// SIMATIC STEP 7 (V5.x) project Daysil_Autoclav_v3

SYMBOL_TABLE
"AI-SENSOR-DATA"	DB 1	DB 1
"ORTAK_DATA"	DB 2	DB 2	// Ortak Veriler
"TIME_OTO_1_DB"	DB 5	SFB 4
"TIME_OTO_2_DB"	DB 6	SFB 4
"TIME_OTO_1_PROSES_DB"	DB 7	SFB 4
"TIME_OTO_2_PROSES_DB"	DB 8	SFB 4
"SURELER_DB"	DB 14	FB 3
"SAFETY_DB"	DB 15	FB 2
"KAZAN1_DATA"	DB 17	DB 17
"KAZAN2_DATA"	DB 18	DB 18	// KAZAN 2 BILGILERI
"JEN1_DATA"	DB 19	DB 19
"JEN2_DATA"	DB 20	DB 20
"JEN1_PID_DATA"	DB 21	DB 21
"JEN2_PID_DATA"	DB 22	DB 22
"KAZAN1_PID_DATA"	DB 23	DB 23	// KAZAN 1 PID BILGILERI
"KAZAN2_PID_DATA"	DB 24	DB 24	// KAZAN 2 PID BILGILERI
"JEN2_KONTROL_BLOGU_DB"	DB 51	FB 50
"JEN_1_PID_DB"	DB 69	FB 58
"JEN_2_PID_DB"	DB 70	FB 58
"OTOKLAV_1_DB"	DB 94	FB 94
"OTOKLAV_2_DB"	DB 95	FB 95
"FB98_DB"	DB 98	FB 98
"FB99_DB"	DB 99	FB 99
"HMI_DATA"	DB 100	DB 100	// Hmi arayuz verileri
"KAZAN_1_PID_DB"	DB 130	FB 58
"KAZAN_2_PID_DATA"	DB 231	FB 58
"MAINBLOCK"	FB 1	FB 1	// ANA PROGRAM BLOGU
"SAFETY"	FB 2	FB 2
"SURELER"	FB 3	FB 3
"TEST_BLOGU"	FB 5	FB 5
"KAZAN_ORTAK"	FB 20	FB 20
"KAZAN_PID_ORTAK"	FB 21	FB 21
"CONT_C"	FB 41	FB 41	// Continuous Control
"KAZAN_1_PID_KONTROL"	FB 47	FB 47
"KAZAN_2_PID_KONTROL"	FB 48	FB 48
"JEN1_PID_KONTROL"	FB 49	FB 49
"JEN2_PID_KONTROL"	FB 50	FB 50	// BUAHR JENERATÖR 2 PID
"TCONT_CP"	FB 58	FB 58	// temperature PID controller with pulse generator and self-tuning
"KAZAN_1_KONTROL"	FB 94	FB 94
"KAZAN_2_KONTROL"	FB 95	FB 95
"KAZAN1_KONTROL_BLOGU"	FB 96	FB 96
"KAZAN2_KONTROL_BLOGU"	FB 97	FB 97
"JEN1_KONTROL_BLOGU"	FB 98	FB 98
"JEN2_KONTROL_BLOGU"	FB 99	FB 99
"TIME_UNSCALE"	FC 1	FC 1
"O.Vana_AciklikHesaplama"	FC 2	FC 2	// Oransal vana aciklik orani hesaplama
"Int_To_S5Time"	FC 10	FC 10
"TIM_S5TI"	FC 40	FC 40	// IEC Time to S5 Time
"SCALE"	FC 105	FC 105	// Scaling Values
"UNSCALE"	FC 106	FC 106	// Unscaling Values
"KAZAN1_ACIL_STOP"	I 0.0	BOOL	// Acil Stop
"KAZAN1_START"	I 0.1	BOOL	// Kazan 1 Start
"KAZAN1_TRANSFER"	I 0.2	BOOL	// Kazan 1 Buhar Transferi
"KAZAN1_BOSALTIM"	I 0.3	BOOL	// Kazan 1 Bosaltim
"KAZAN1_KAPAK_SW"	I 0.4	BOOL	// Kazan 1 Kapak Kapandi
"KAZAN2_ACIL_STOP"	I 0.5	BOOL	// Kazan 2 Acil Stop
"KAZAN2_START"	I 0.6	BOOL	// Kazan 2 Start
"KAZAN2_TRANSFER"	I 0.7	BOOL	// Kazan 2 Buhar Transferi
"KAZAN2_BOSALTIM"	I 1.0	BOOL	// Kazan 2 Bosaltim
"KAZAN2_KAPAK_SW"	I 1.1	BOOL	// Kazan 2 Kapak Kapandi
"JEN1_STOP"	I 1.2	BOOL	// Jenerator 1 Stop
"JEN1_START"	I 1.3	BOOL	// Jenerator 1 Start
"JEN2_STOP"	I 1.4	BOOL	// Jenerator 2 Stop
"JEN2_START"	I 1.5	BOOL	// Jenerator 2 Start
"MANUEL"	I 1.6	BOOL	// Manuel Mod
"OTOMATIK"	I 1.7	BOOL	// Otomatik Mod
"JEN2_MOTOR_CALISTI"	I 2.0	BOOL
"JEN_1_MIN_SU_SEVIYESI"	I 3.0	BOOL
"JEN_2_MIN_SU_SEVIYESI"	I 3.1	BOOL
"0.1 SN."	M 0.0	BOOL
"0.2 SN."	M 0.1	BOOL
"0.4 SN."	M 0.2	BOOL
"0.5 SN."	M 0.3	BOOL
"0.8 SN."	M 0.4	BOOL
"1.0 SN."	M 0.5	BOOL
"1.6 SN."	M 0.6	BOOL
"2.0 SN."	M 0.7	BOOL
"Oto_1_Proses_BASLADI"	M 20.0	BOOL
"Oto_2_Proses_Basladi"	M 20.1	BOOL
"JEN2_CALIS_SURESI_BASLA"	M 22.0	BOOL
"JEN2_CALISTI_RIS"	M 22.1	BOOL
"JEN1_CALIS_SURESI_BASLA"	M 23.0	BOOL
"JEN1_CALISTI_RIS"	M 23.1	BOOL
"Jen1_Guvenlik_set_reset"	M 25.0	BOOL
"Jen2_Guvenlik_Set_Reset"	M 26.0	BOOL
"OTO_1_BEKLEME_BASLADI"	M 27.0	BOOL
"OTO_2_BEKLEME_BASLADI"	M 27.1	BOOL
"KAZAN_1_PID_MAN_ON"	M 35.0	BOOL
"KAZAN_2_MAN_ON"	M 37.0	BOOL
"TEST_START"	M 40.0	BOOL
"TEST_STOP"	M 40.1	BOOL
"TEST_OUT"	M 40.2	BOOL
"ALWAYS OFF"	M 100.0	BOOL	// ALWAYS OFF
"ALWAYS ON"	M 100.1	BOOL	// ALWAYS ON
"SET2_ULASMADI_SR"	M 101.0	BOOL
"SET2_ULASMADI_RIS"	M 101.1	BOOL
"JEN2_TCONT_MAN_ON"	M 155.0	BOOL
"Jen2_Stop_Trigger"	M 200.0	BOOL
"Jen2_Stop_Ris"	M 200.1	BOOL
"Jen2_Stop_Set_Mem"	M 200.2	BOOL
"JEN2_STOP_SET_RESET"	M 201.0	BOOL
"Sicaklik Dustu"	M 201.1	BOOL
"Ris_Jen2_Sicaklik_Dustu"	M 201.2	BOOL
"Rising_Sogutma"	M 201.3	BOOL
"Falling_Sogutma"	M 201.4	BOOL
"JEN1_STOP_SET_RESET"	M 202.0	BOOL
"START"	M 700.1	BOOL
"PID_START"	M 700.2	BOOL
"BRULOR_START"	M 700.3	BOOL
"SICAKLIK_1_OK"	M 700.5	BOOL
"SICAKLIK_2_OK"	M 700.6	BOOL
"BURLOR_MOTOR_START"	M 700.7	BOOL
"STOP"	M 701.1	BOOL
"100_DERECE_RIS"	M 750.0	BOOL
"Jen2_Ris"	M 750.4	BOOL
"Jen1_Ris"	M 750.5	BOOL
"BOS"	M 1000.0	BOOL
"O.VanaIlkAciklik"	MD 42	REAL	// Oransal vana ilk aciklik orani
"O.VanaKademeArtis"	MD 46	REAL	// Oransal vana kademeli artis orani
"PID BLOCK"	OB 35	OB 35	// PID BLOCK
"ZAMANHATASI"	OB 80	OB 80	// ZAMAN HATASI
"GERILIMHATASI"	OB 81	OB 81	// BESLEME GERILIMI HATASI
"HATAUYARISI"	OB 82	OB 82	// HATA UYARISI
"TAKMACIKARMAHATASI"	OB 83	OB 83	// TAKMA ÇIKARMA UYARISI
"CPUHARDWAREERROR"	OB 84	OB 84	// CPU HARDWARE ERROR
"PROGRAMHATASI"	OB 85	OB 85	// PROGRAM YURUTME HATASI
"RACKHATASI"	OB 86	OB 86	// RACK HATASI
"HABERLESMEHATASI"	OB 87	OB 87	// HABERLESME HATASI,
"COMPLETE RESTART"	OB 100	OB 100	// Complete Restart
"RESTART"	OB 101	OB 101	// Restart
"COLD RESTART"	OB 102	OB 102	// Cold Restart
"PROGRAMMINGERROR"	OB 121	OB 121	// PROGRAMLAMA HATASI
"MOD_ERR"	OB 122	OB 122	// Module Access Error
"KAZAN1_YESIL_LAMBA"	Q 0.0	BOOL	// Kazan 1 Yesil Lamba
"KAZAN1_KIRMIZI_LAMBA"	Q 0.1	BOOL	// Kazan 1 Kirmizi Lamba
"KAZAN1_DUDUK"	Q 0.2	BOOL	// Kazan 1 Duduk
"KAZAN1_BOSALTIM_VALFI"	Q 0.3	BOOL	// Kazan 1 Buhar Bosaltim
"KAZAN1_TRANS_BUT_LAMBASI"	Q 0.4	BOOL	// Kazan 1 Transfer Lambasi
"KAZAN1_EMN_VALFI_BOS"	Q 0.5	BOOL	// Kazan  1 Emniyet vantili bosaltim valfi
"KAZAN2_YESIL_LAMBA"	Q 0.6	BOOL	// Kazan 2 Yesil Lamba
"KAZAN2_KIRMIZI_LAMBA"	Q 0.7	BOOL	// Kazan 2 Kirmizi Lamba
"KAZAN2_DUDUK"	Q 1.0	BOOL	// Kazan 2 Duduk
"KAZAN2_BOSALTIM_VALFI"	Q 1.1	BOOL	// Kazan 2 Buhar Bosaltim
"KAZAN2_TRANS_BUT_LAMBASI"	Q 1.2	BOOL	// Kazan 2 Transfer Lambasi
"KAZAN2_EMN_VALFI_BOS"	Q 1.3	BOOL	// Kazan Emniyet vantili bosaltim valfi
"JEN_1_HAT_VANASI"	Q 1.4	BOOL
"JEN_1_PANO_STOP_LAMBASI"	Q 1.5	BOOL
"JEN_1_PANO_START_LAMBASI"	Q 1.6	BOOL
"JEN_2_HAT_VANASI"	Q 1.7	BOOL
"JEN_2_PANO_STOP_LAMBASI"	Q 2.0	BOOL
"JEN_2_PANO_START_LAMBASI"	Q 2.1	BOOL
"PANO_OTO_MAN_BUTON_LAMBA"	Q 2.2	BOOL
"PANO_ALARM"	Q 2.3	BOOL
"JEN_1_BRULOR"	Q 2.4	BOOL
"JEN_1_POMPA"	Q 2.5	BOOL
"JEN_2_BRULOR_OUT"	Q 2.6	BOOL
"JEN_2_SU_POM_OUT"	Q 2.7	BOOL
"TON"	SFB 4	SFB 4	// Generate an On Delay
"TIME_TCK"	SFC 64	SFC 64	// Read the System Time
"delay_300ms_1"	T 8	TIMER
"500ms_delay1"	T 10	TIMER
"1s Delay"	T 11	TIMER
"Pisim_Suresi"	T 12	TIMER
"500ms_delay"	T 13	TIMER
"s_offt_7s_delay"	T 14	TIMER
"tm_adim1_pid_basla_delay"	T 16	TIMER
"500ms_delay_kazan_2"	T 20	TIMER
"1ms_delay_kazan_2"	T 21	TIMER
"kazan_2_pisirme_delay"	T 22	TIMER
"kazan_2_500ms_delay"	T 23	TIMER
"kazan_2_7s_delay"	T 24	TIMER
"Delay_500ms_Jen2"	T 30	TIMER
"DELAY_1S_JEN_HATA"	T 33	TIMER
"DELAY_300MS"	T 42	TIMER
"DELAY_500MS_1"	T 43	TIMER
"DELAY_5S_pompa"	T 44	TIMER
"OTO_2_DELAY_BITIS"	T 50	TIMER
"OTO_1_DELAY_PISIM_BITTI"	T 51	TIMER
"DELAY_ADIM5_BEKLE"	T 52	TIMER
"DELAY_ADIM5_BEKLE2"	T 53	TIMER
"TIM_SET2_ULASMADI"	T 57	TIMER
"VAT_1"	VAT 1	
END_SYMBOL_TABLE

FUNCTION_BLOCK "MAINBLOCK"	// FB 1
VERSION : 0.1
BEGIN
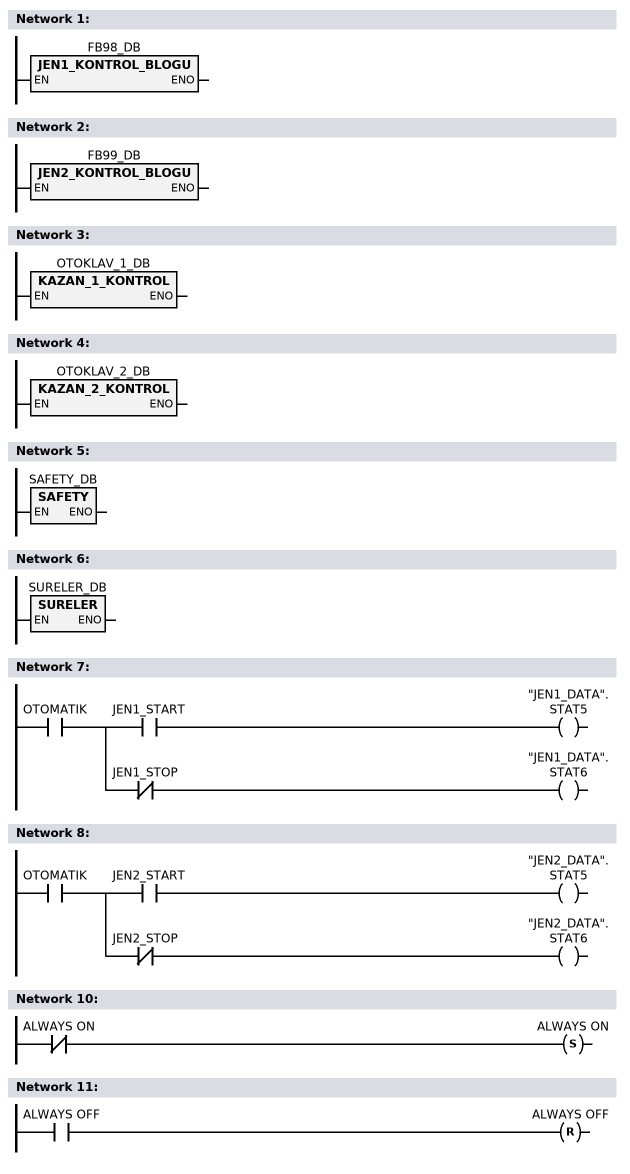
NETWORK
TITLE =
      CALL  "JEN1_KONTROL_BLOGU" , "FB98_DB";
      NOP   0;
NETWORK
TITLE =
      CALL  "JEN2_KONTROL_BLOGU" , "FB99_DB";
      NOP   0;
NETWORK
TITLE =
      CALL  "KAZAN_1_KONTROL" , "OTOKLAV_1_DB";
      NOP   0;
NETWORK
TITLE =
      CALL  "KAZAN_2_KONTROL" , "OTOKLAV_2_DB";
      NOP   0;
NETWORK
TITLE =
      CALL  "SAFETY" , "SAFETY_DB";
      NOP   0;
NETWORK
TITLE =
      CALL  "SURELER" , "SURELER_DB";
      NOP   0;
NETWORK
TITLE =
      A     "OTOMATIK";
      =     L 0.0;
      A     L 0.0;
      A     "JEN1_START";
      =     "JEN1_DATA".STAT5;
      A     L 0.0;
      AN    "JEN1_STOP";
      =     "JEN1_DATA".STAT6;
NETWORK
TITLE =
      A     "OTOMATIK";
      =     L 0.0;
      A     L 0.0;
      A     "JEN2_START";
      =     "JEN2_DATA".STAT5;
      A     L 0.0;
      AN    "JEN2_STOP";
      =     "JEN2_DATA".STAT6;
NETWORK
TITLE =
NETWORK
TITLE =
      AN    "ALWAYS ON";
      S     "ALWAYS ON";
NETWORK
TITLE =
      A     "ALWAYS OFF";
      R     "ALWAYS OFF";
NETWORK
TITLE =
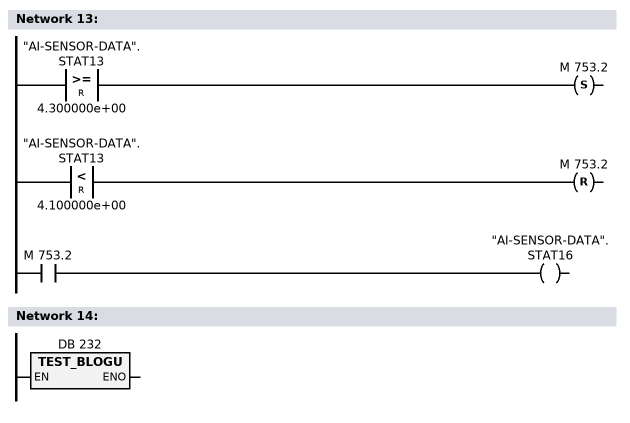
NETWORK
TITLE =
      A(;
      L     "AI-SENSOR-DATA".STAT13;
      L     4.300000e+00;
      >=R;
      );
      S     M 753.2;
      A(;
      L     "AI-SENSOR-DATA".STAT13;
      L     4.100000e+00;
      <R;
      );
      R     M 753.2;
      A     M 753.2;
      =     "AI-SENSOR-DATA".STAT16;
NETWORK
TITLE =
      CALL  "TEST_BLOGU" , DB 232;
      NOP   0;
END_FUNCTION_BLOCK

FUNCTION_BLOCK "SAFETY"	// FB 2
VERSION : 0.1
BEGIN
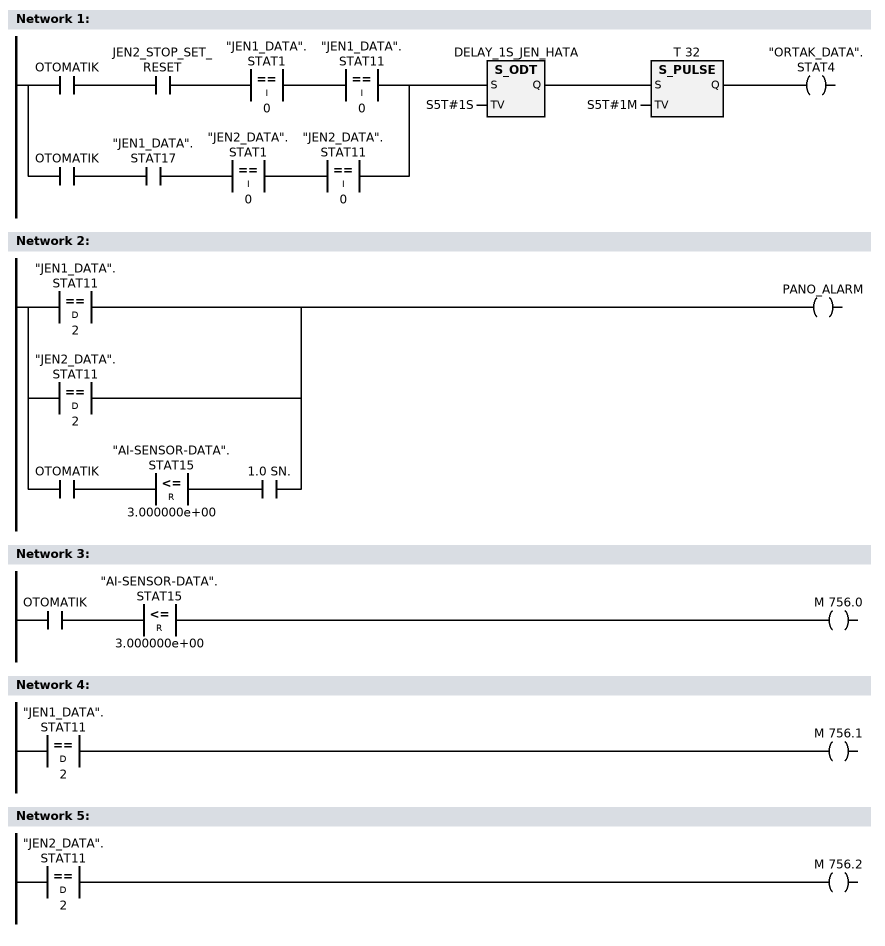
NETWORK
TITLE =
      A(;
      A(;
      A     "OTOMATIK";
      A     "JEN2_STOP_SET_RESET";
      A(;
      L     "JEN1_DATA".STAT1;
      L     0;
      ==I;
      );
      A(;
      L     "JEN1_DATA".STAT11;
      L     0;
      ==I;
      );
      O;
      A     "OTOMATIK";
      A     "JEN1_DATA".STAT17;
      A(;
      L     "JEN2_DATA".STAT1;
      L     0;
      ==I;
      );
      A(;
      L     "JEN2_DATA".STAT11;
      L     0;
      ==I;
      );
      );
      L     S5T#1S;
      SD    "DELAY_1S_JEN_HATA";
      NOP   0;
      NOP   0;
      NOP   0;
      A     "DELAY_1S_JEN_HATA";
      );
      L     S5T#1M;
      SP    T 32;
      NOP   0;
      NOP   0;
      NOP   0;
      A     T 32;
      =     "ORTAK_DATA".STAT4;
NETWORK
TITLE =
      O(;
      L     "JEN1_DATA".STAT11;
      L     2;
      ==D;
      );
      O(;
      L     "JEN2_DATA".STAT11;
      L     2;
      ==D;
      );
      O;
      A     "OTOMATIK";
      A(;
      L     "AI-SENSOR-DATA".STAT15;
      L     3.000000e+00;
      <=R;
      );
      A     "1.0 SN.";
      =     "PANO_ALARM";
NETWORK
TITLE =
      A     "OTOMATIK";
      A(;
      L     "AI-SENSOR-DATA".STAT15;
      L     3.000000e+00;
      <=R;
      );
      =     M 756.0;
NETWORK
TITLE =
      L     "JEN1_DATA".STAT11;
      L     2;
      ==D;
      =     M 756.1;
NETWORK
TITLE =
      L     "JEN2_DATA".STAT11;
      L     2;
      ==D;
      =     M 756.2;
END_FUNCTION_BLOCK

FUNCTION_BLOCK "SURELER"	// FB 3
VERSION : 0.1
BEGIN
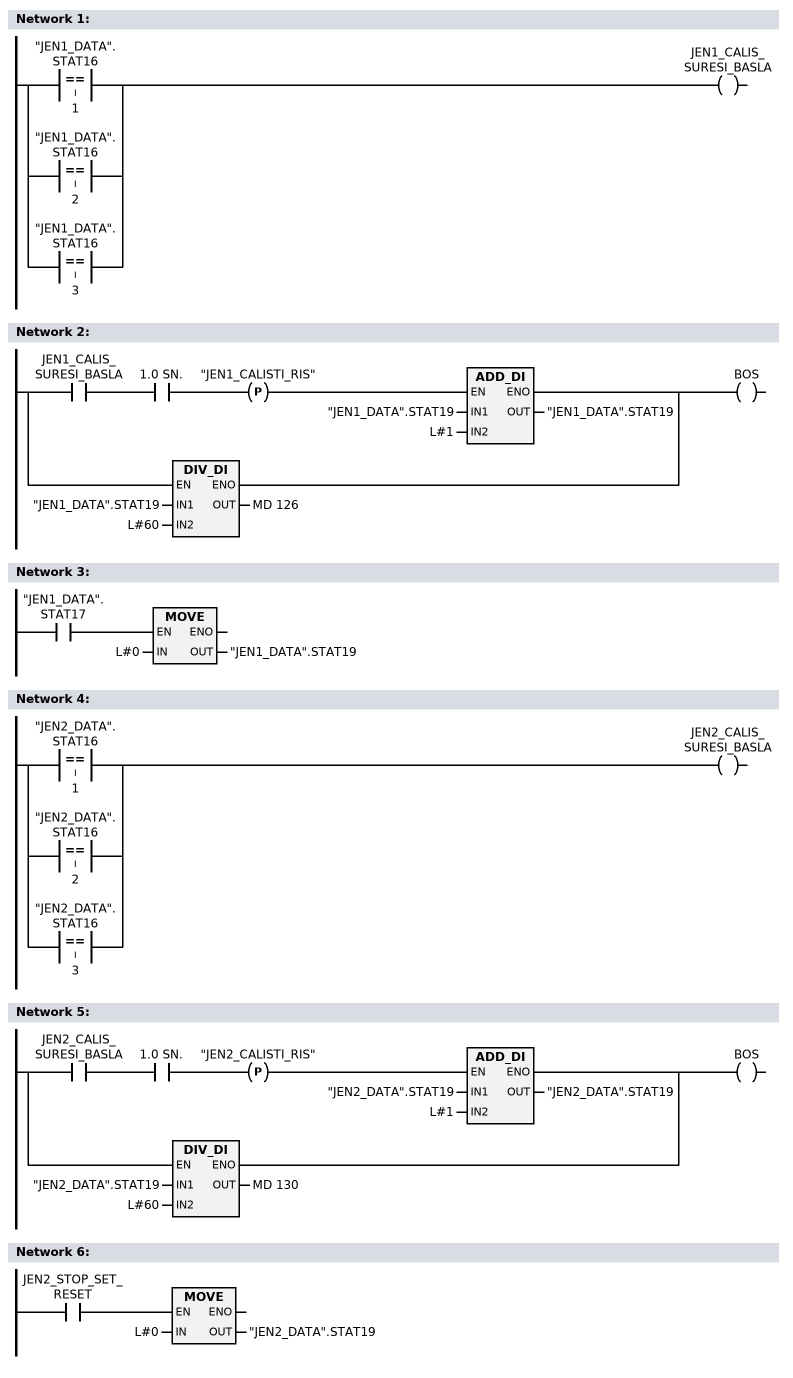
NETWORK
TITLE =
      O(;
      L     "JEN1_DATA".STAT16;
      L     1;
      ==I;
      );
      O(;
      L     "JEN1_DATA".STAT16;
      L     2;
      ==I;
      );
      O(;
      L     "JEN1_DATA".STAT16;
      L     3;
      ==I;
      );
      =     "JEN1_CALIS_SURESI_BASLA";
NETWORK
TITLE =
      O(;
      A     "JEN1_CALIS_SURESI_BASLA";
      A     "1.0 SN.";
      FP    "JEN1_CALISTI_RIS";
      JNB   _001;
      L     "JEN1_DATA".STAT19;
      L     L#1;
      +D;
      T     "JEN1_DATA".STAT19;
      AN    OV;
      SAVE;
      CLR;
_001: A     BR;
      );
      O(;
      L     "JEN1_DATA".STAT19;
      L     L#60;
      /D;
      T     MD 126;
      AN    OV;
      SAVE;
      CLR;
      A     BR;
      );
      =     "BOS";
NETWORK
TITLE =
      A     "JEN1_DATA".STAT17;
      JNB   _002;
      L     L#0;
      T     "JEN1_DATA".STAT19;
_002: NOP   0;
NETWORK
TITLE =
      O(;
      L     "JEN2_DATA".STAT16;
      L     1;
      ==I;
      );
      O(;
      L     "JEN2_DATA".STAT16;
      L     2;
      ==I;
      );
      O(;
      L     "JEN2_DATA".STAT16;
      L     3;
      ==I;
      );
      =     "JEN2_CALIS_SURESI_BASLA";
NETWORK
TITLE =
      O(;
      A     "JEN2_CALIS_SURESI_BASLA";
      A     "1.0 SN.";
      FP    "JEN2_CALISTI_RIS";
      JNB   _003;
      L     "JEN2_DATA".STAT19;
      L     L#1;
      +D;
      T     "JEN2_DATA".STAT19;
      AN    OV;
      SAVE;
      CLR;
_003: A     BR;
      );
      O(;
      L     "JEN2_DATA".STAT19;
      L     L#60;
      /D;
      T     MD 130;
      AN    OV;
      SAVE;
      CLR;
      A     BR;
      );
      =     "BOS";
NETWORK
TITLE =
      A     "JEN2_STOP_SET_RESET";
      JNB   _004;
      L     L#0;
      T     "JEN2_DATA".STAT19;
_004: NOP   0;
NETWORK
TITLE =
      O(;
      A(;
      A     "KAZAN1_DATA".STAT19;
      =     L 0.0;
      BLD   103;
      BLD   9;
      =     L 5.0;
      CDB;
      OPN   DI 5;
      TAR2  LD 1;
      A     L 0.0;
      =     DIX 0.0;
      L     L#82800000;
      T     DID 2;
      LAR2  P#DBX 0.0;
      UC    "TON";
      LAR2  LD 1;
      L     DID 8;
      OPN   DI 17;
      T     DID 42;
      OPN   DI 5;
      CDB;
      BLD   10;
      A     BR;
      );
      JNB   _005;
      CALL  "TIME_UNSCALE" (
           $1                       := "KAZAN1_DATA".STAT20,
           $2                       := "KAZAN1_DATA".STAT3,
           $3                       := "KAZAN1_DATA".STAT21);
_005: A     BR;
      );
      O(;
      L     "KAZAN1_DATA".STAT21;
      L     60;
      /D;
      T     MD 118;
      AN    OV;
      SAVE;
      CLR;
      A     BR;
      );
      =     "BOS";
NETWORK
TITLE =
      O(;
      A(;
      A     "KAZAN2_DATA".STAT19;
      =     L 0.0;
      BLD   103;
      BLD   9;
      =     L 5.0;
      CDB;
      OPN   DI 6;
      TAR2  LD 1;
      A     L 0.0;
      =     DIX 0.0;
      L     L#82800000;
      T     DID 2;
      LAR2  P#DBX 0.0;
      UC    "TON";
      LAR2  LD 1;
      L     DID 8;
      OPN   DI 18;
      T     DID 42;
      OPN   DI 6;
      CDB;
      BLD   10;
      A     BR;
      );
      JNB   _006;
      CALL  "TIME_UNSCALE" (
           $1                       := "KAZAN2_DATA".STAT20,
           $2                       := "KAZAN2_DATA".STAT3,
           $3                       := "KAZAN2_DATA".STAT21);
_006: A     BR;
      );
      O(;
      L     "KAZAN2_DATA".STAT21;
      L     60;
      /D;
      T     MD 122;
      AN    OV;
      SAVE;
      CLR;
      A     BR;
      );
      =     "BOS";
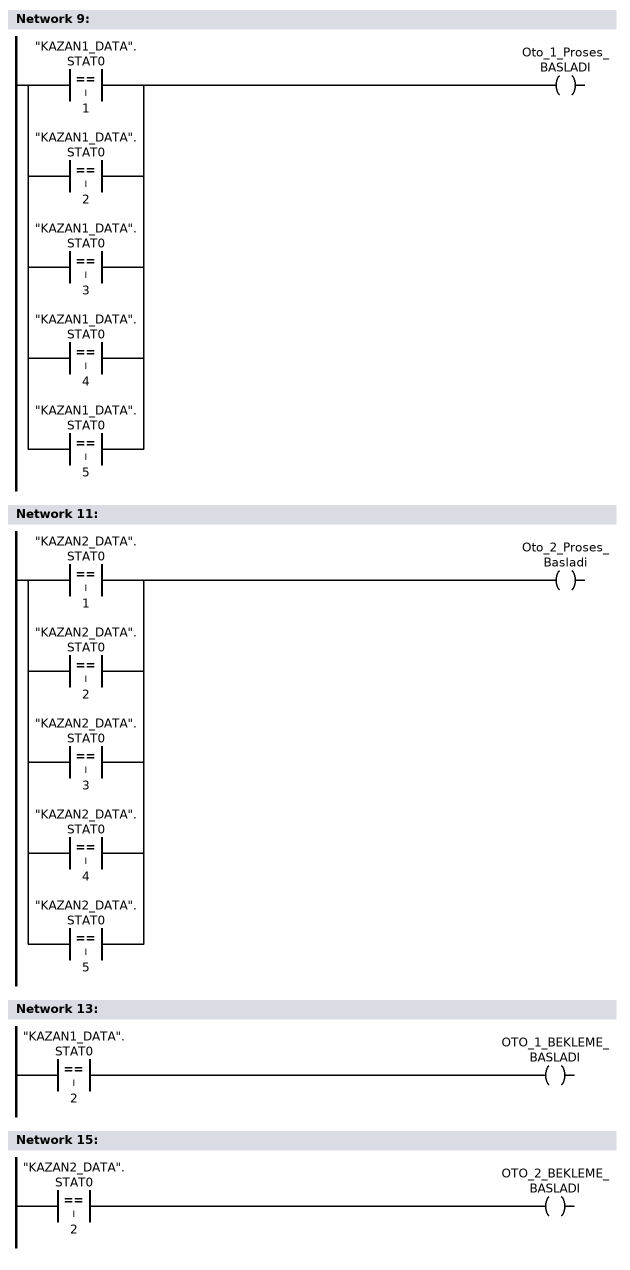
NETWORK
TITLE =
      O(;
      L     "KAZAN1_DATA".STAT0;
      L     1;
      ==I;
      );
      O(;
      L     "KAZAN1_DATA".STAT0;
      L     2;
      ==I;
      );
      O(;
      L     "KAZAN1_DATA".STAT0;
      L     3;
      ==I;
      );
      O(;
      L     "KAZAN1_DATA".STAT0;
      L     4;
      ==I;
      );
      O(;
      L     "KAZAN1_DATA".STAT0;
      L     5;
      ==I;
      );
      =     "Oto_1_Proses_BASLADI";
NETWORK
TITLE =
      O(;
      A(;
      A     "Oto_1_Proses_BASLADI";
      =     L 0.0;
      BLD   103;
      BLD   9;
      =     L 5.0;
      CDB;
      OPN   DI 7;
      TAR2  LD 1;
      A     L 0.0;
      =     DIX 0.0;
      L     L#82800000;
      T     DID 2;
      LAR2  P#DBX 0.0;
      UC    "TON";
      LAR2  LD 1;
      L     DID 8;
      OPN   DI 17;
      T     DID 50;
      OPN   DI 7;
      CDB;
      BLD   10;
      A     BR;
      );
      JNB   _007;
      L     "KAZAN1_DATA".STAT22;
      L     1000;
      /D;
      T     "KAZAN1_DATA".STAT23;
      AN    OV;
      SAVE;
      CLR;
_007: A     BR;
      );
      O(;
      L     "KAZAN1_DATA".STAT23;
      L     60;
      /D;
      T     MD 110;
      AN    OV;
      SAVE;
      CLR;
      A     BR;
      );
      =     "BOS";
NETWORK
TITLE =
      O(;
      L     "KAZAN2_DATA".STAT0;
      L     1;
      ==I;
      );
      O(;
      L     "KAZAN2_DATA".STAT0;
      L     2;
      ==I;
      );
      O(;
      L     "KAZAN2_DATA".STAT0;
      L     3;
      ==I;
      );
      O(;
      L     "KAZAN2_DATA".STAT0;
      L     4;
      ==I;
      );
      O(;
      L     "KAZAN2_DATA".STAT0;
      L     5;
      ==I;
      );
      =     "Oto_2_Proses_Basladi";
NETWORK
TITLE =
      O(;
      A(;
      A     "Oto_2_Proses_Basladi";
      =     L 0.0;
      BLD   103;
      BLD   9;
      =     L 5.0;
      CDB;
      OPN   DI 8;
      TAR2  LD 1;
      A     L 0.0;
      =     DIX 0.0;
      L     L#82800000;
      T     DID 2;
      LAR2  P#DBX 0.0;
      UC    "TON";
      LAR2  LD 1;
      L     DID 8;
      OPN   DI 18;
      T     DID 50;
      OPN   DI 8;
      CDB;
      BLD   10;
      A     BR;
      );
      JNB   _008;
      L     "KAZAN2_DATA".STAT22;
      L     1000;
      /D;
      T     "KAZAN2_DATA".STAT23;
      AN    OV;
      SAVE;
      CLR;
_008: A     BR;
      );
      O(;
      L     "KAZAN2_DATA".STAT23;
      L     60;
      /D;
      T     MD 114;
      AN    OV;
      SAVE;
      CLR;
      A     BR;
      );
      =     "BOS";
NETWORK
TITLE =
      L     "KAZAN1_DATA".STAT0;
      L     2;
      ==I;
      =     "OTO_1_BEKLEME_BASLADI";
NETWORK
TITLE =
      A(;
      A     "OTO_1_BEKLEME_BASLADI";
      =     L 0.0;
      BLD   103;
      BLD   9;
      =     L 5.0;
      CDB;
      OPN   DI 9;
      TAR2  LD 1;
      A     L 0.0;
      =     DIX 0.0;
      L     L#82800000;
      T     DID 2;
      LAR2  P#DBX 0.0;
      UC    "TON";
      LAR2  LD 1;
      L     DID 8;
      OPN   DI 17;
      T     DID 58;
      OPN   DI 9;
      CDB;
      BLD   10;
      A     BR;
      );
      JNB   _009;
      L     "KAZAN1_DATA".STAT24;
      L     1000;
      /D;
      T     "KAZAN1_DATA".STAT25;
_009: NOP   0;
NETWORK
TITLE =
      L     "KAZAN2_DATA".STAT0;
      L     2;
      ==I;
      =     "OTO_2_BEKLEME_BASLADI";
NETWORK
TITLE =
      A(;
      A     "OTO_2_BEKLEME_BASLADI";
      =     L 0.0;
      BLD   103;
      BLD   9;
      =     L 5.0;
      CDB;
      OPN   DI 10;
      TAR2  LD 1;
      A     L 0.0;
      =     DIX 0.0;
      L     L#82800000;
      T     DID 2;
      LAR2  P#DBX 0.0;
      UC    "TON";
      LAR2  LD 1;
      L     DID 8;
      OPN   DI 18;
      T     DID 58;
      OPN   DI 10;
      CDB;
      BLD   10;
      A     BR;
      );
      JNB   _00a;
      L     "KAZAN2_DATA".STAT24;
      L     1000;
      /D;
      T     "KAZAN2_DATA".STAT25;
_00a: NOP   0;
END_FUNCTION_BLOCK

FUNCTION_BLOCK "TEST_BLOGU"	// FB 5
VERSION : 0.1
BEGIN
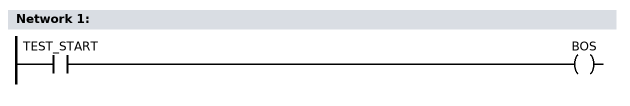
NETWORK
TITLE =
      A     "TEST_START";
      =     "BOS";
END_FUNCTION_BLOCK

FUNCTION_BLOCK "KAZAN_ORTAK"	// FB 20
VERSION : 0.1
VAR_INPUT
  IN0 : BOOL ;
  IN1 : BOOL ;
  IN2 : BOOL ;
  IN3 : BOOL ;
  IN4 : BOOL ;
  IN5 : BOOL ;
  IN6 : BOOL ;
  IN7 : BOOL ;
  IN8 : BOOL ;
  IN9 : S5TIME ;
  IN10 : INT ;
  IN11 : REAL ;
  IN12 : REAL ;
  IN13 : TIMER ;
  IN14 : TIMER ;
  IN15 : TIMER ;
  IN16 : TIMER ;
  IN17 : TIMER ;
  IN18 : REAL ;
  IN19 : REAL ;
  IN20 : REAL ;
  IN21 : REAL ;
  IN22 : INT ;
  IN23 : BOOL ;
  IN24 : BOOL ;
  IN25 : BLOCK_DB ;
  IN26 : BOOL ;
  IN27 : BOOL ;
  IN28 : REAL ;
  IN29 : TIMER ;
  IN30 : TIMER ;
  IN31 : TIMER ;
  IN32 : TIMER ;
END_VAR
VAR_OUTPUT
  OUT33 : BOOL ;
  OUT34 : BOOL ;
  OUT35 : BOOL ;
  OUT36 : BOOL ;
  OUT37 : BOOL ;
  OUT38 : REAL ;
  OUT39 : BOOL ;
  OUT40 : WORD ;
  OUT41 : REAL ;
  OUT42 : BOOL ;
  OUT43 : BOOL ;
  OUT44 : WORD ;
  OUT45 : REAL ;
  OUT46 : BOOL ;
  OUT47 : BOOL ;
  OUT48 : BOOL ;
  OUT49 : BOOL ;
END_VAR
VAR_IN_OUT
  IO50 : INT ;
END_VAR
VAR
  STAT51 : INT ;
  STAT52 : BOOL ;
  STAT53 : BOOL ;
  STAT54 : REAL ;
  STAT55 : BOOL ;
  STAT56 : REAL  := 1.000000e+001;
  STAT57 : REAL ;
  STAT58 : BOOL ;
  STAT59 : REAL ;
  STAT60 : REAL ;
  STAT61 : BOOL ;
  STAT62 : BOOL ;
  STAT63 : BOOL ;
  STAT64 : BOOL ;
  STAT65 : WORD ;
  STAT66 : REAL ;
  STAT67 : WORD ;
  STAT68 : REAL ;
  STAT69 : BOOL ;
  STAT70 : BOOL ;
  STAT71 : BOOL ;
  STAT72 : REAL ;
  STAT73 : TIME ;
  STAT74 : BOOL ;
  STAT75 : BOOL ;
  STAT76 : BOOL ;
  STAT77 : BOOL ;
  STAT78 : BOOL ;
END_VAR
VAR_TEMP
  tKademe : STRUCT
   Bir : REAL ;
   Iki : REAL ;
   Uc : REAL ;
   Dort : REAL ;
   Bes : REAL ;
   Alti : REAL ;
   Yedi : REAL ;
  END_STRUCT ;
END_VAR
BEGIN
NETWORK
TITLE =
      A(;
      A(;
      A     "ALWAYS OFF";
      =     L 28.0;
      BLD   103;
      CALL  "SCALE" (
           $1                       := #IN10,
           $2                       := #IN18,
           $3                       := #IN19,
           $4                       := L 28.0,
           $5                       := #STAT65,
           $6                       := #STAT66);
      A     BR;
      );
      JNB   _001;
      L     #STAT65;
      T     #OUT40;
      SET;
      SAVE;
      CLR;
_001: A     BR;
      );
      JNB   _002;
      L     #STAT66;
      T     #OUT41;
_002: NOP   0;
NETWORK
TITLE =
      A(;
      A(;
      A     "ALWAYS OFF";
      =     L 28.0;
      BLD   103;
      CALL  "SCALE" (
           $1                       := #IN22,
           $2                       := #IN20,
           $3                       := #IN21,
           $4                       := L 28.0,
           $5                       := #STAT67,
           $6                       := #STAT68);
      A     BR;
      );
      JNB   _003;
      L     #STAT67;
      T     #OUT44;
      SET;
      SAVE;
      CLR;
_003: A     BR;
      );
      JNB   _004;
      L     #STAT68;
      T     #OUT45;
_004: NOP   0;
NETWORK
TITLE =
      A(;
      A     "OTOMATIK";
      A     #IN0;
      A     "AI-SENSOR-DATA".STAT16;
      L     S5T#200MS;
      T     LD 28;
      TAK;
      T     LD 32;
      L     #IN13;
      T     LW 36;
      L     LD 32;
      L     LD 28;
      SD    T [LW 36];
      NOP   0;
      NOP   0;
      NOP   0;
      T     LD 28;
      TAK;
      T     LD 32;
      L     #IN13;
      T     LW 36;
      L     LD 32;
      L     LD 28;
      A     T [LW 36];
      );
      A     #IN4;
      A     #IN1;
      A(;
      L     #IO50;
      L     0;
      ==I;
      );
      JNB   _005;
      L     1;
      T     #IO50;
      SET;
      SAVE;
      CLR;
_005: A     BR;
      S     #STAT69;
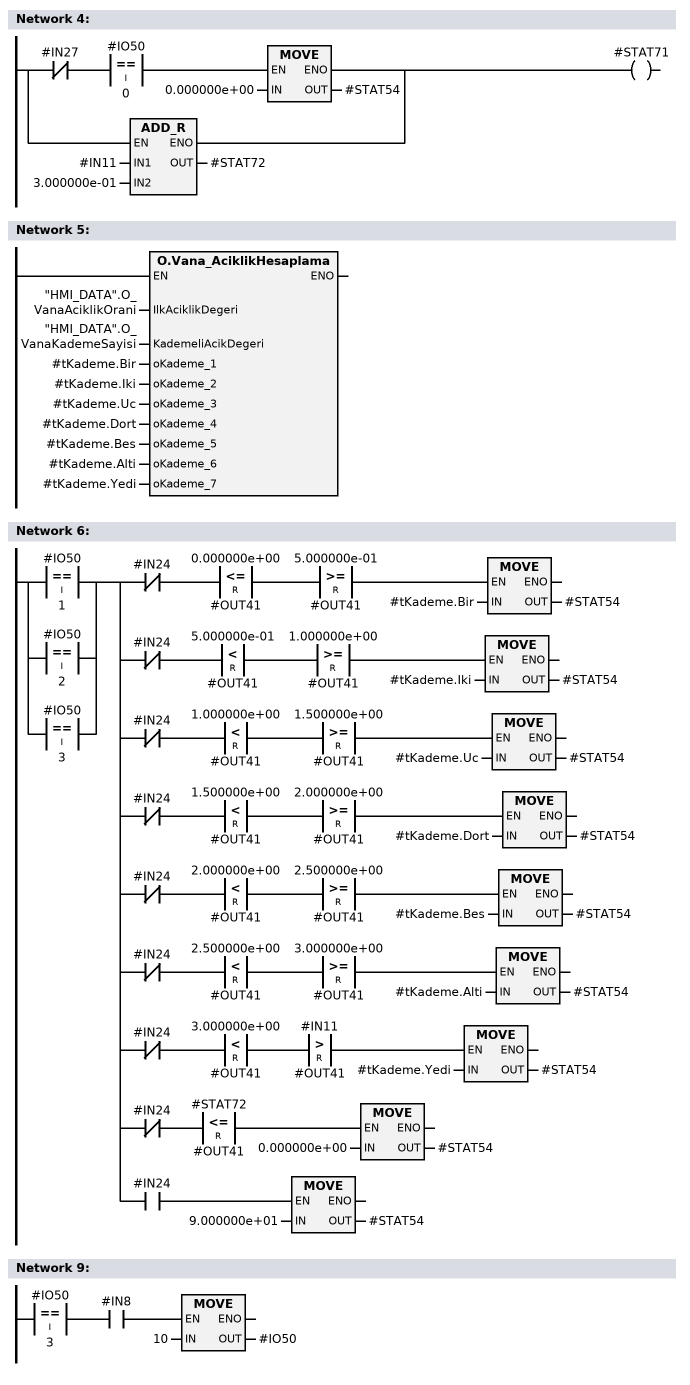
NETWORK
TITLE =
      O(;
      AN    #IN27;
      A(;
      L     #IO50;
      L     0;
      ==I;
      );
      JNB   _006;
      L     0.000000e+00;
      T     #STAT54;
      SET;
      SAVE;
      CLR;
_006: A     BR;
      );
      O(;
      L     #IN11;
      L     3.000000e-01;
      +R;
      T     #STAT72;
      AN    OV;
      SAVE;
      CLR;
      A     BR;
      );
      =     #STAT71;
NETWORK
TITLE =
      CALL  "O.Vana_AciklikHesaplama" (
           IlkAciklikDegeri         := "HMI_DATA".O_VanaAciklikOrani,
           KademeliAcikDegeri       := "HMI_DATA".O_VanaKademeSayisi,
           oKademe_1                := #tKademe.Bir,
           oKademe_2                := #tKademe.Iki,
           oKademe_3                := #tKademe.Uc,
           oKademe_4                := #tKademe.Dort,
           oKademe_5                := #tKademe.Bes,
           oKademe_6                := #tKademe.Alti,
           oKademe_7                := #tKademe.Yedi);
      NOP   0;
NETWORK
TITLE =
      O(;
      L     #IO50;
      L     1;
      ==I;
      );
      O(;
      L     #IO50;
      L     2;
      ==I;
      );
      O(;
      L     #IO50;
      L     3;
      ==I;
      );
      =     L 28.0;
      A     L 28.0;
      AN    #IN24;
      A(;
      L     0.000000e+00;
      L     #OUT41;
      <=R;
      );
      A(;
      L     5.000000e-01;
      L     #OUT41;
      >=R;
      );
      JNB   _007;
      L     #tKademe.Bir;
      T     #STAT54;
_007: NOP   0;
      A     L 28.0;
      AN    #IN24;
      A(;
      L     5.000000e-01;
      L     #OUT41;
      <R;
      );
      A(;
      L     1.000000e+00;
      L     #OUT41;
      >=R;
      );
      JNB   _008;
      L     #tKademe.Iki;
      T     #STAT54;
_008: NOP   0;
      A     L 28.0;
      AN    #IN24;
      A(;
      L     1.000000e+00;
      L     #OUT41;
      <R;
      );
      A(;
      L     1.500000e+00;
      L     #OUT41;
      >=R;
      );
      JNB   _009;
      L     #tKademe.Uc;
      T     #STAT54;
_009: NOP   0;
      A     L 28.0;
      AN    #IN24;
      A(;
      L     1.500000e+00;
      L     #OUT41;
      <R;
      );
      A(;
      L     2.000000e+00;
      L     #OUT41;
      >=R;
      );
      JNB   _00a;
      L     #tKademe.Dort;
      T     #STAT54;
_00a: NOP   0;
      A     L 28.0;
      AN    #IN24;
      A(;
      L     2.000000e+00;
      L     #OUT41;
      <R;
      );
      A(;
      L     2.500000e+00;
      L     #OUT41;
      >=R;
      );
      JNB   _00b;
      L     #tKademe.Bes;
      T     #STAT54;
_00b: NOP   0;
      A     L 28.0;
      AN    #IN24;
      A(;
      L     2.500000e+00;
      L     #OUT41;
      <R;
      );
      A(;
      L     3.000000e+00;
      L     #OUT41;
      >=R;
      );
      JNB   _00c;
      L     #tKademe.Alti;
      T     #STAT54;
_00c: NOP   0;
      A     L 28.0;
      AN    #IN24;
      A(;
      L     3.000000e+00;
      L     #OUT41;
      <R;
      );
      A(;
      L     #IN11;
      L     #OUT41;
      >R;
      );
      JNB   _00d;
      L     #tKademe.Yedi;
      T     #STAT54;
_00d: NOP   0;
      A     L 28.0;
      AN    #IN24;
      A(;
      L     #STAT72;
      L     #OUT41;
      <=R;
      );
      JNB   _00e;
      L     0.000000e+00;
      T     #STAT54;
_00e: NOP   0;
      A     L 28.0;
      A     #IN24;
      JNB   _00f;
      L     9.000000e+01;
      T     #STAT54;
_00f: NOP   0;
NETWORK
TITLE =
      L     #IO50;
      L     1;
      ==I;
      =     L 28.0;
      A(;
      A     L 28.0;
      A     #STAT58;
      L     #IN9;
      T     LD 29;
      TAK;
      T     LD 33;
      L     #IN15;
      T     LW 37;
      L     LD 33;
      L     LD 29;
      SD    T [LW 37];
      NOP   0;
      NOP   0;
      NOP   0;
      T     LD 29;
      TAK;
      T     LD 33;
      L     #IN15;
      T     LW 37;
      L     LD 33;
      L     LD 29;
      A     T [LW 37];
      );
      JNB   _010;
      L     2;
      T     #IO50;
_010: NOP   0;
      A     L 28.0;
      A(;
      O(;
      L     #OUT41;
      L     #IN11;
      >=R;
      );
      O     #STAT58;
      );
      =     #STAT58;
NETWORK
TITLE =
      L     #IO50;
      L     2;
      ==I;
      =     L 28.0;
      A     L 28.0;
      L     S5T#5M;
      T     LD 29;
      TAK;
      T     LD 33;
      L     #IN31;
      T     LW 37;
      L     LD 33;
      L     LD 29;
      SD    T [LW 37];
      NOP   0;
      NOP   0;
      NOP   0;
      NOP   0;
      A     L 28.0;
      A     #IN2;
      JNB   _011;
      L     3;
      T     #IO50;
_011: NOP   0;
      A     L 28.0;
      A     #IN3;
      JNB   _012;
      L     4;
      T     #IO50;
_012: NOP   0;
NETWORK
TITLE =
      A(;
      L     #IO50;
      L     3;
      ==I;
      );
      A     #IN8;
      JNB   _013;
      L     10;
      T     #IO50;
_013: NOP   0;
NETWORK
TITLE =
      L     #IO50;
      L     10;
      ==I;
      =     L 28.0;
      A     L 28.0;
      JNB   _014;
      L     9.000000e+01;
      T     #STAT54;
      SET;
      SAVE;
      CLR;
_014: A     BR;
      =     #OUT39;
      A(;
      A     L 28.0;
      L     S5T#23S;
      T     LD 29;
      TAK;
      T     LD 33;
      L     #IN16;
      T     LW 37;
      L     LD 33;
      L     LD 29;
      SD    T [LW 37];
      NOP   0;
      NOP   0;
      NOP   0;
      T     LD 29;
      TAK;
      T     LD 33;
      L     #IN16;
      T     LW 37;
      L     LD 33;
      L     LD 29;
      A     T [LW 37];
      );
      JNB   _015;
      L     4;
      T     #IO50;
_015: NOP   0;
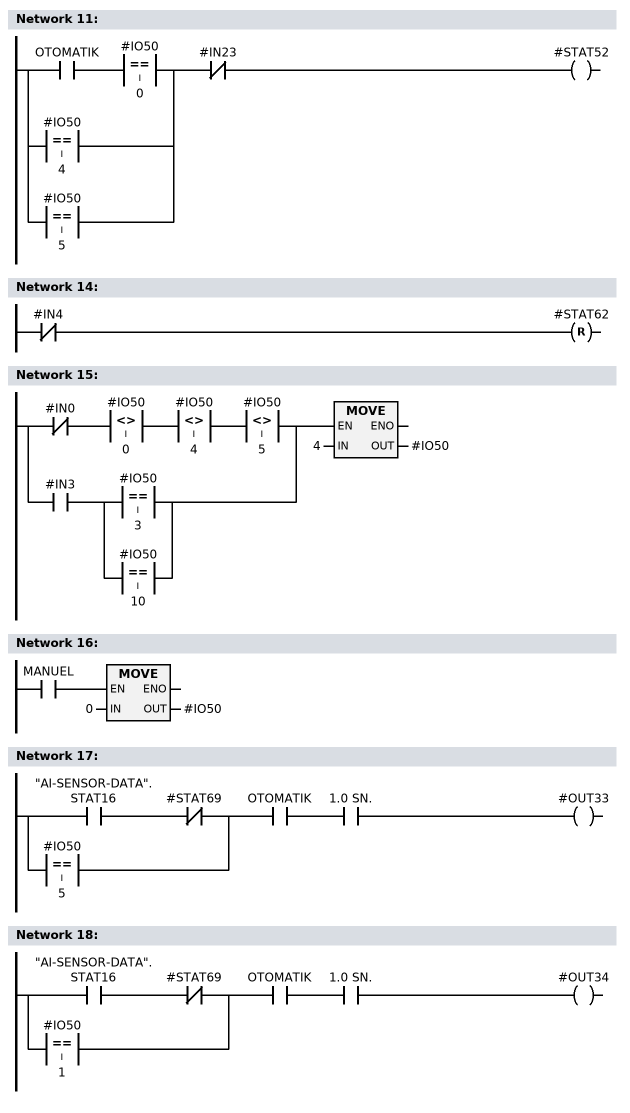
NETWORK
TITLE =
      A(;
      A     "OTOMATIK";
      A(;
      L     #IO50;
      L     0;
      ==I;
      );
      O(;
      L     #IO50;
      L     4;
      ==I;
      );
      O(;
      L     #IO50;
      L     5;
      ==I;
      );
      );
      AN    #IN23;
      =     #STAT52;
NETWORK
TITLE =
      L     #IO50;
      L     4;
      ==I;
      =     L 28.0;
      A     L 28.0;
      JNB   _016;
      L     0.000000e+00;
      T     #STAT54;
_016: NOP   0;
      A     L 28.0;
      BLD   102;
      =     #STAT70;
      A     L 28.0;
      A(;
      L     #OUT41;
      L     1.000000e-01;
      <=R;
      );
      =     L 28.1;
      A     L 28.1;
      BLD   102;
      S     #STAT62;
      A(;
      A     L 28.1;
      L     S5T#5S;
      T     LD 29;
      TAK;
      T     LD 33;
      L     #IN29;
      T     LW 37;
      L     LD 33;
      L     LD 29;
      SD    T [LW 37];
      NOP   0;
      NOP   0;
      NOP   0;
      T     LD 29;
      TAK;
      T     LD 33;
      L     #IN29;
      T     LW 37;
      L     LD 33;
      L     LD 29;
      A     T [LW 37];
      );
      JNB   _017;
      L     5;
      T     #IO50;
_017: NOP   0;
NETWORK
TITLE =
      A(;
      A(;
      L     #IO50;
      L     5;
      ==I;
      );
      L     S5T#1S;
      T     LD 28;
      TAK;
      T     LD 32;
      L     #IN30;
      T     LW 36;
      L     LD 32;
      L     LD 28;
      SD    T [LW 36];
      NOP   0;
      NOP   0;
      NOP   0;
      T     LD 28;
      TAK;
      T     LD 32;
      L     #IN30;
      T     LW 36;
      L     LD 32;
      L     LD 28;
      A     T [LW 36];
      );
      AN    #IN4;
      JNB   _018;
      L     0;
      T     #IO50;
_018: NOP   0;
NETWORK
TITLE =
      AN    #IN4;
      R     #STAT62;
NETWORK
TITLE =
      A(;
      AN    #IN0;
      A(;
      L     #IO50;
      L     0;
      <>I;
      );
      A(;
      L     #IO50;
      L     4;
      <>I;
      );
      A(;
      L     #IO50;
      L     5;
      <>I;
      );
      O;
      A     #IN3;
      A(;
      O(;
      L     #IO50;
      L     3;
      ==I;
      );
      O(;
      L     #IO50;
      L     10;
      ==I;
      );
      );
      );
      JNB   _019;
      L     4;
      T     #IO50;
_019: NOP   0;
NETWORK
TITLE =
      A     "MANUEL";
      JNB   _01a;
      L     0;
      T     #IO50;
_01a: NOP   0;
NETWORK
TITLE =
      A(;
      A     "AI-SENSOR-DATA".STAT16;
      AN    #STAT69;
      O(;
      L     #IO50;
      L     5;
      ==I;
      );
      );
      A     "OTOMATIK";
      A     "1.0 SN.";
      =     #OUT33;
NETWORK
TITLE =
      A(;
      A     "AI-SENSOR-DATA".STAT16;
      AN    #STAT69;
      O(;
      L     #IO50;
      L     1;
      ==I;
      );
      );
      A     "OTOMATIK";
      A     "1.0 SN.";
      =     #OUT34;
NETWORK
TITLE =
      A(;
      A(;
      L     #IO50;
      L     2;
      ==I;
      );
      A     "1.0 SN.";
      O(;
      A(;
      O(;
      L     #IO50;
      L     3;
      ==I;
      );
      O(;
      L     #IO50;
      L     10;
      ==I;
      );
      );
      AN    #OUT39;
      L     S5T#5M;
      T     LD 28;
      TAK;
      T     LD 32;
      L     #IN32;
      T     LW 36;
      L     LD 32;
      L     LD 28;
      SD    T [LW 36];
      NOP   0;
      NOP   0;
      NOP   0;
      T     LD 28;
      TAK;
      T     LD 32;
      L     #IN32;
      T     LW 36;
      L     LD 32;
      L     LD 28;
      A     T [LW 36];
      );
      );
      A     "OTOMATIK";
      =     #OUT35;
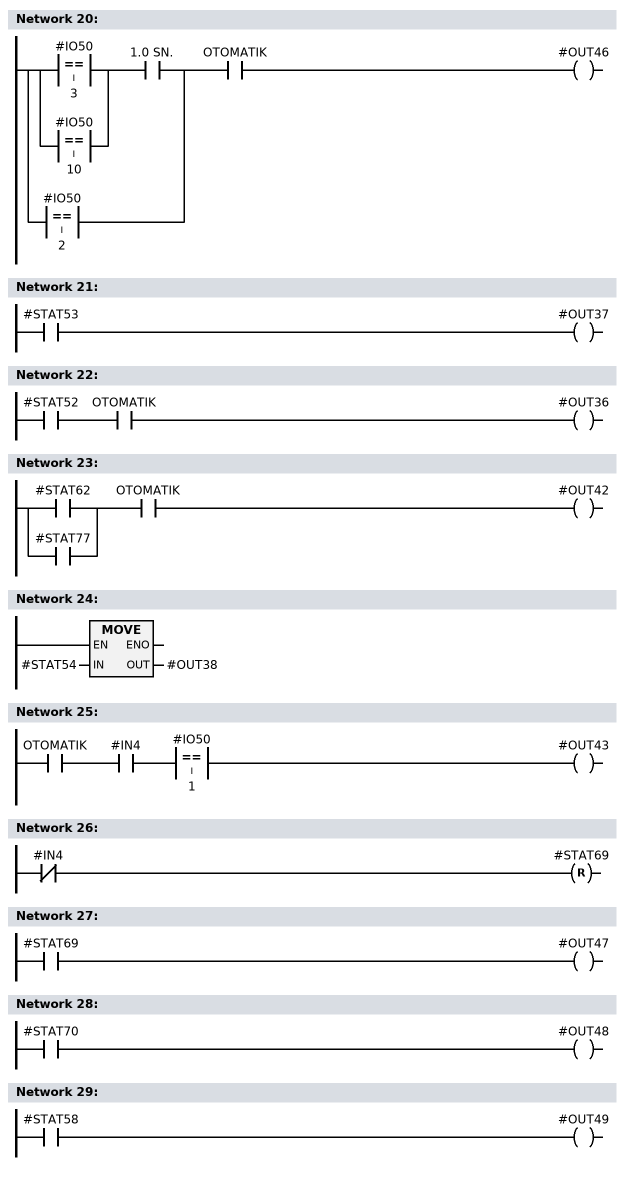
NETWORK
TITLE =
      A(;
      A(;
      O(;
      L     #IO50;
      L     3;
      ==I;
      );
      O(;
      L     #IO50;
      L     10;
      ==I;
      );
      );
      A     "1.0 SN.";
      O(;
      L     #IO50;
      L     2;
      ==I;
      );
      );
      A     "OTOMATIK";
      =     #OUT46;
NETWORK
TITLE =
      A     #STAT53;
      =     #OUT37;
NETWORK
TITLE =
      A     #STAT52;
      A     "OTOMATIK";
      =     #OUT36;
NETWORK
TITLE =
      A(;
      O     #STAT62;
      O     #STAT77;
      );
      A     "OTOMATIK";
      =     #OUT42;
NETWORK
TITLE =
      L     #STAT54;
      T     #OUT38;
      NOP   0;
NETWORK
TITLE =
      A     "OTOMATIK";
      A     #IN4;
      A(;
      L     #IO50;
      L     1;
      ==I;
      );
      =     #OUT43;
NETWORK
TITLE =
      AN    #IN4;
      R     #STAT69;
NETWORK
TITLE =
      A     #STAT69;
      =     #OUT47;
NETWORK
TITLE =
      A     #STAT70;
      =     #OUT48;
NETWORK
TITLE =
      A     #STAT58;
      =     #OUT49;
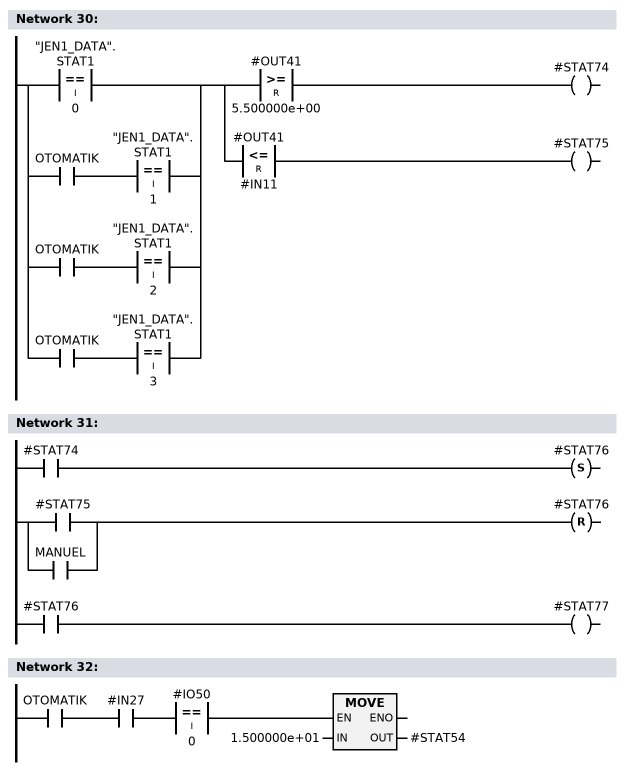
NETWORK
TITLE =
      O(;
      L     "JEN1_DATA".STAT1;
      L     0;
      ==I;
      );
      O;
      A     "OTOMATIK";
      A(;
      L     "JEN1_DATA".STAT1;
      L     1;
      ==I;
      );
      O;
      A     "OTOMATIK";
      A(;
      L     "JEN1_DATA".STAT1;
      L     2;
      ==I;
      );
      O;
      A     "OTOMATIK";
      A(;
      L     "JEN1_DATA".STAT1;
      L     3;
      ==I;
      );
      =     L 28.0;
      A     L 28.0;
      A(;
      L     #OUT41;
      L     5.500000e+00;
      >=R;
      );
      =     #STAT74;
      A     L 28.0;
      A(;
      L     #OUT41;
      L     #IN11;
      <=R;
      );
      =     #STAT75;
NETWORK
TITLE =
      A     #STAT74;
      S     #STAT76;
      A(;
      O     #STAT75;
      O     "MANUEL";
      );
      R     #STAT76;
      A     #STAT76;
      =     #STAT77;
NETWORK
TITLE =
      A     "OTOMATIK";
      A     #IN27;
      A(;
      L     #IO50;
      L     0;
      ==I;
      );
      JNB   _01b;
      L     1.500000e+01;
      T     #STAT54;
_01b: NOP   0;
END_FUNCTION_BLOCK

// FB 41: know-how protected block, not included

FUNCTION_BLOCK "KAZAN_1_PID_KONTROL"	// FB 47
VERSION : 0.1
BEGIN
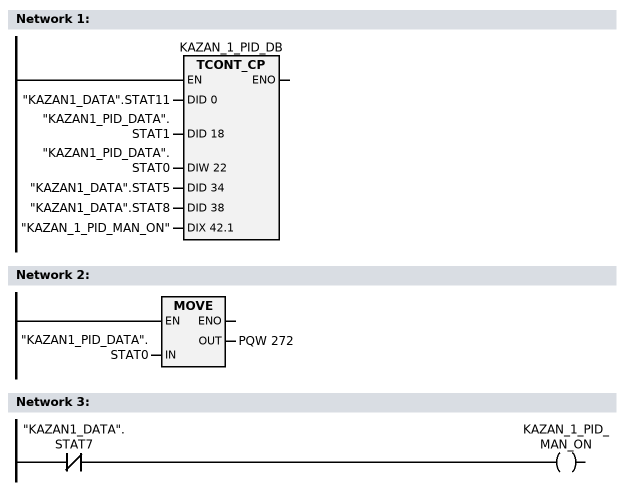
NETWORK
TITLE =
      CALL  "TCONT_CP" , "KAZAN_1_PID_DB" (
           DID 0                    := "KAZAN1_DATA".STAT11,
           DID 18                   := "KAZAN1_PID_DATA".STAT1,
           DIW 22                   := "KAZAN1_PID_DATA".STAT0,
           DID 34                   := "KAZAN1_DATA".STAT5,
           DID 38                   := "KAZAN1_DATA".STAT8,
           DIX 42.1                 := "KAZAN_1_PID_MAN_ON");
      NOP   0;
NETWORK
TITLE =
      L     "KAZAN1_PID_DATA".STAT0;
      T     PQW 272;
      NOP   0;
NETWORK
TITLE =
      AN    "KAZAN1_DATA".STAT7;
      =     "KAZAN_1_PID_MAN_ON";
NETWORK
TITLE =
END_FUNCTION_BLOCK

FUNCTION_BLOCK "KAZAN_2_PID_KONTROL"	// FB 48
VERSION : 0.1
BEGIN
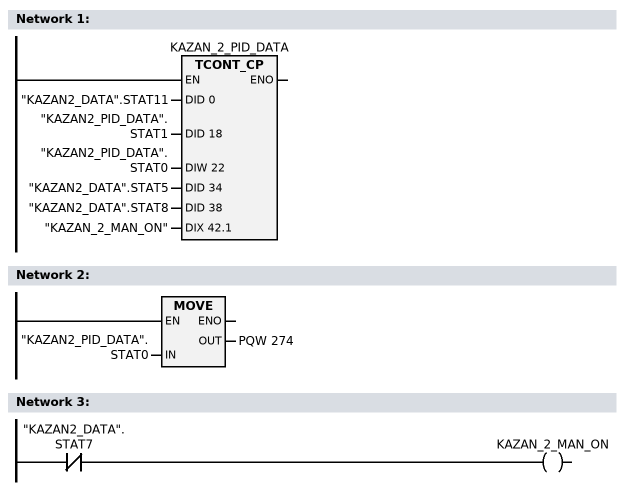
NETWORK
TITLE =
      CALL  "TCONT_CP" , "KAZAN_2_PID_DATA" (
           DID 0                    := "KAZAN2_DATA".STAT11,
           DID 18                   := "KAZAN2_PID_DATA".STAT1,
           DIW 22                   := "KAZAN2_PID_DATA".STAT0,
           DID 34                   := "KAZAN2_DATA".STAT5,
           DID 38                   := "KAZAN2_DATA".STAT8,
           DIX 42.1                 := "KAZAN_2_MAN_ON");
      NOP   0;
NETWORK
TITLE =
      L     "KAZAN2_PID_DATA".STAT0;
      T     PQW 274;
      NOP   0;
NETWORK
TITLE =
      AN    "KAZAN2_DATA".STAT7;
      =     "KAZAN_2_MAN_ON";
END_FUNCTION_BLOCK

FUNCTION_BLOCK "JEN1_PID_KONTROL"	// FB 49
VERSION : 0.1
VAR
  STAT0 : REAL ;
  STAT1 : BOOL ;
  STAT2 : REAL ;
  STAT3 : INT ;
END_VAR
BEGIN
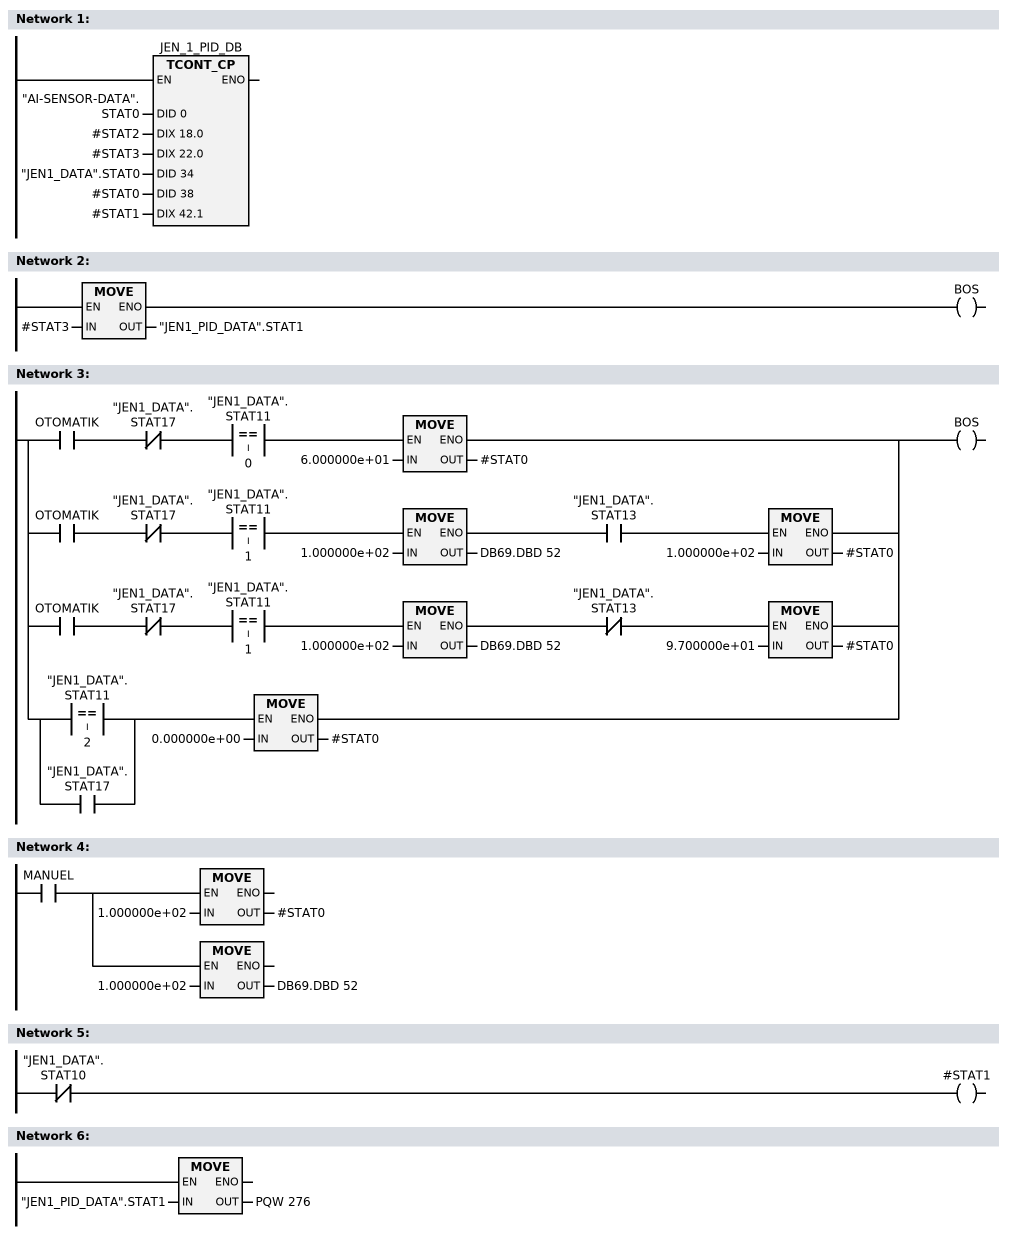
NETWORK
TITLE =
      CALL  "TCONT_CP" , "JEN_1_PID_DB" (
           DID 0                    := "AI-SENSOR-DATA".STAT0,
           DIX 18.0                 := #STAT2,
           DIX 22.0                 := #STAT3,
           DID 34                   := "JEN1_DATA".STAT0,
           DID 38                   := #STAT0,
           DIX 42.1                 := #STAT1);
      NOP   0;
NETWORK
TITLE =
      L     #STAT3;
      T     "JEN1_PID_DATA".STAT1;
      SET;
      SAVE;
      CLR;
      A     BR;
      =     "BOS";
NETWORK
TITLE =
      O(;
      A     "OTOMATIK";
      AN    "JEN1_DATA".STAT17;
      A(;
      L     "JEN1_DATA".STAT11;
      L     0;
      ==I;
      );
      JNB   _001;
      L     6.000000e+01;
      T     #STAT0;
      SET;
      SAVE;
      CLR;
_001: A     BR;
      );
      O(;
      A(;
      A     "OTOMATIK";
      AN    "JEN1_DATA".STAT17;
      A(;
      L     "JEN1_DATA".STAT11;
      L     1;
      ==I;
      );
      JNB   _002;
      L     1.000000e+02;
      T     DB69.DBD 52;
      SET;
      SAVE;
      CLR;
_002: A     BR;
      );
      A     "JEN1_DATA".STAT13;
      JNB   _003;
      L     1.000000e+02;
      T     #STAT0;
      SET;
      SAVE;
      CLR;
_003: A     BR;
      );
      O(;
      A(;
      A     "OTOMATIK";
      AN    "JEN1_DATA".STAT17;
      A(;
      L     "JEN1_DATA".STAT11;
      L     1;
      ==I;
      );
      JNB   _004;
      L     1.000000e+02;
      T     DB69.DBD 52;
      SET;
      SAVE;
      CLR;
_004: A     BR;
      );
      AN    "JEN1_DATA".STAT13;
      JNB   _005;
      L     9.700000e+01;
      T     #STAT0;
      SET;
      SAVE;
      CLR;
_005: A     BR;
      );
      O(;
      A(;
      O(;
      L     "JEN1_DATA".STAT11;
      L     2;
      ==I;
      );
      O     "JEN1_DATA".STAT17;
      );
      JNB   _006;
      L     0.000000e+00;
      T     #STAT0;
      SET;
      SAVE;
      CLR;
_006: A     BR;
      );
      =     "BOS";
NETWORK
TITLE =
      A     "MANUEL";
      =     L 0.0;
      A     L 0.0;
      JNB   _007;
      L     1.000000e+02;
      T     #STAT0;
_007: NOP   0;
      A     L 0.0;
      JNB   _008;
      L     1.000000e+02;
      T     DB69.DBD 52;
_008: NOP   0;
NETWORK
TITLE =
      AN    "JEN1_DATA".STAT10;
      =     #STAT1;
NETWORK
TITLE =
      L     "JEN1_PID_DATA".STAT1;
      T     PQW 276;
      NOP   0;
END_FUNCTION_BLOCK

FUNCTION_BLOCK "JEN2_PID_KONTROL"	// FB 50
VERSION : 0.1
VAR
  STAT0 : REAL ;
  STAT1 : INT ;
  STAT2 : REAL ;
  STAT3 : BOOL ;
  STAT4 : BOOL ;
END_VAR
BEGIN
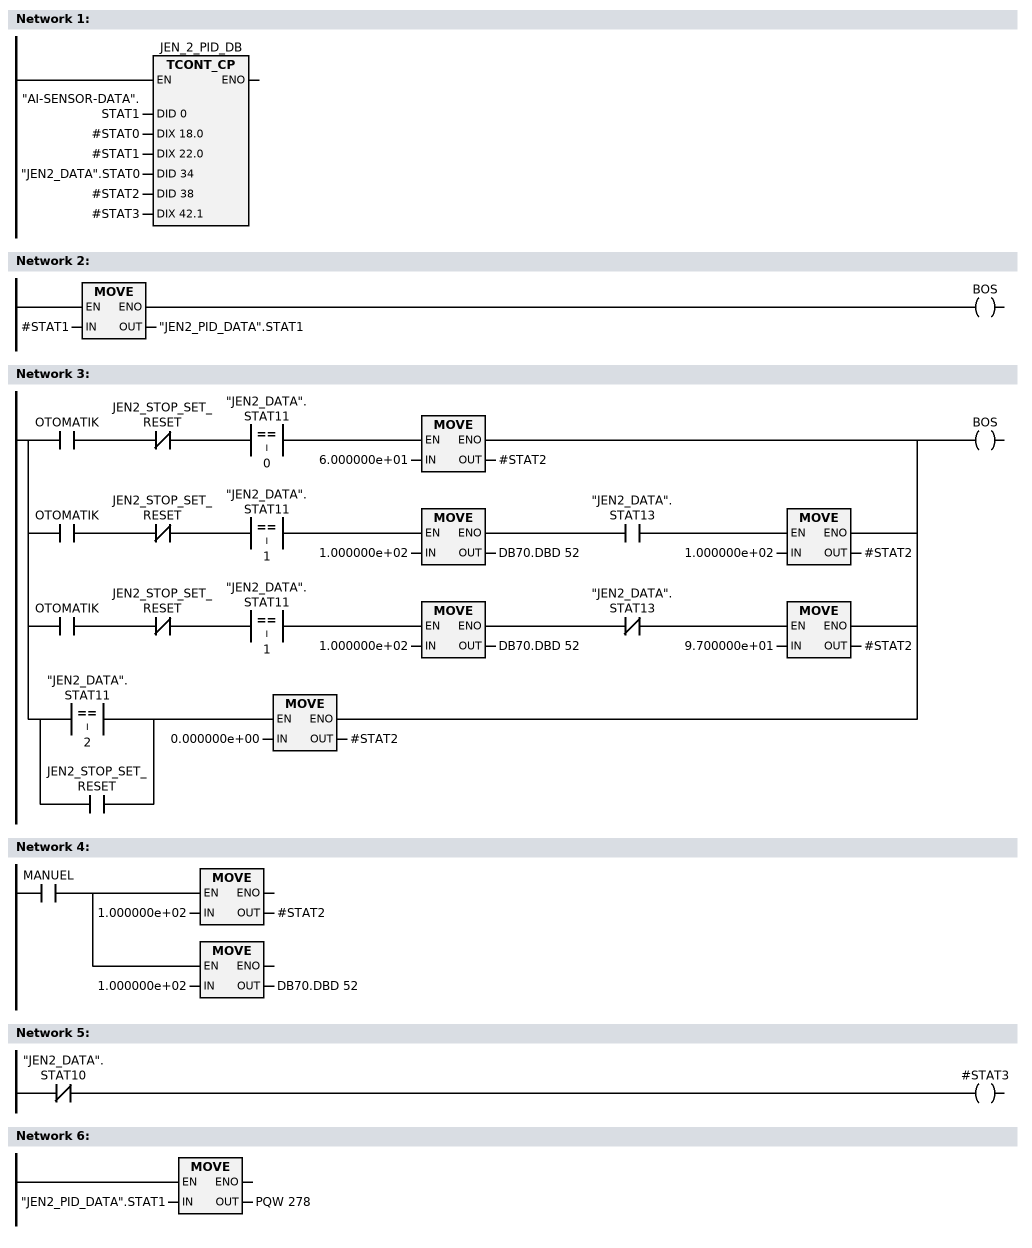
NETWORK
TITLE =
      CALL  "TCONT_CP" , "JEN_2_PID_DB" (
           DID 0                    := "AI-SENSOR-DATA".STAT1,
           DIX 18.0                 := #STAT0,
           DIX 22.0                 := #STAT1,
           DID 34                   := "JEN2_DATA".STAT0,
           DID 38                   := #STAT2,
           DIX 42.1                 := #STAT3);
      NOP   0;
NETWORK
TITLE =
      L     #STAT1;
      T     "JEN2_PID_DATA".STAT1;
      SET;
      SAVE;
      CLR;
      A     BR;
      =     "BOS";
NETWORK
TITLE =
      O(;
      A     "OTOMATIK";
      AN    "JEN2_STOP_SET_RESET";
      A(;
      L     "JEN2_DATA".STAT11;
      L     0;
      ==I;
      );
      JNB   _001;
      L     6.000000e+01;
      T     #STAT2;
      SET;
      SAVE;
      CLR;
_001: A     BR;
      );
      O(;
      A(;
      A     "OTOMATIK";
      AN    "JEN2_STOP_SET_RESET";
      A(;
      L     "JEN2_DATA".STAT11;
      L     1;
      ==I;
      );
      JNB   _002;
      L     1.000000e+02;
      T     DB70.DBD 52;
      SET;
      SAVE;
      CLR;
_002: A     BR;
      );
      A     "JEN2_DATA".STAT13;
      JNB   _003;
      L     1.000000e+02;
      T     #STAT2;
      SET;
      SAVE;
      CLR;
_003: A     BR;
      );
      O(;
      A(;
      A     "OTOMATIK";
      AN    "JEN2_STOP_SET_RESET";
      A(;
      L     "JEN2_DATA".STAT11;
      L     1;
      ==I;
      );
      JNB   _004;
      L     1.000000e+02;
      T     DB70.DBD 52;
      SET;
      SAVE;
      CLR;
_004: A     BR;
      );
      AN    "JEN2_DATA".STAT13;
      JNB   _005;
      L     9.700000e+01;
      T     #STAT2;
      SET;
      SAVE;
      CLR;
_005: A     BR;
      );
      O(;
      A(;
      O(;
      L     "JEN2_DATA".STAT11;
      L     2;
      ==I;
      );
      O     "JEN2_STOP_SET_RESET";
      );
      JNB   _006;
      L     0.000000e+00;
      T     #STAT2;
      SET;
      SAVE;
      CLR;
_006: A     BR;
      );
      =     "BOS";
NETWORK
TITLE =
      A     "MANUEL";
      =     L 0.0;
      A     L 0.0;
      JNB   _007;
      L     1.000000e+02;
      T     #STAT2;
_007: NOP   0;
      A     L 0.0;
      JNB   _008;
      L     1.000000e+02;
      T     DB70.DBD 52;
_008: NOP   0;
NETWORK
TITLE =
      AN    "JEN2_DATA".STAT10;
      =     #STAT3;
NETWORK
TITLE =
      L     "JEN2_PID_DATA".STAT1;
      T     PQW 278;
      NOP   0;
END_FUNCTION_BLOCK

// FB 58: know-how protected block, not included

FUNCTION_BLOCK "KAZAN_1_KONTROL"	// FB 94
VERSION : 0.1
BEGIN
NETWORK
TITLE =
      CALL  "Int_To_S5Time" (
           Saat                     := "HMI_DATA".Otoklav_1_TimeData.Hours,
           Dakika                   := "HMI_DATA".Otoklav_1_TimeData.Minutes,
           HesaplananSure_S5TIME    := "KAZAN1_DATA".STAT3);
      CALL  "KAZAN_ORTAK" , DB 120 (
           IN0                      := "KAZAN1_ACIL_STOP",
           IN1                      := "KAZAN1_START",
           IN2                      := "KAZAN1_TRANSFER",
           IN3                      := "KAZAN1_BOSALTIM",
           IN4                      := "KAZAN1_KAPAK_SW",
           IN7                      := "KAZAN1_DATA".STAT1,
           IN8                      := "KAZAN1_DATA".STAT2,
           IN9                      := "KAZAN1_DATA".STAT3,
           IN10                     := "KAZAN1_DATA".STAT4,
           IN11                     := "KAZAN1_DATA".STAT5,
           IN12                     := "KAZAN1_DATA".STAT6,
           IN13                     := "500ms_delay1",
           IN14                     := "1s Delay",
           IN15                     := "Pisim_Suresi",
           IN16                     := "500ms_delay",
           IN17                     := "s_offt_7s_delay",
           IN18                     := 1.000000e+01,
           IN19                     := 0.000000e+00,
           IN20                     := 2.000000e+02,
           IN21                     := 0.000000e+00,
           IN22                     := "KAZAN1_DATA".STAT15,
           IN23                     := "KAZAN1_DATA".STAT17,
           IN24                     := "KAZAN1_DATA".STAT18,
           IN27                     := "ORTAK_DATA".STAT4,
           IN29                     := "OTO_1_DELAY_PISIM_BITTI",
           IN30                     := "DELAY_ADIM5_BEKLE",
           IN31                     := T 58,
           IN32                     := T 61,
           OUT33                    := "KAZAN1_YESIL_LAMBA",
           OUT34                    := "KAZAN1_KIRMIZI_LAMBA",
           OUT35                    := "KAZAN1_DUDUK",
           OUT36                    := "KAZAN1_BOSALTIM_VALFI",
           OUT37                    := "KAZAN1_DATA".STAT7,
           OUT38                    := "KAZAN1_DATA".STAT8,
           OUT39                    := "KAZAN1_DATA".STAT9,
           OUT40                    := "KAZAN1_DATA".STAT10,
           OUT41                    := "KAZAN1_DATA".STAT11,
           OUT42                    := "KAZAN1_EMN_VALFI_BOS",
           OUT43                    := "KAZAN1_DATA".STAT12,
           OUT44                    := "KAZAN1_DATA".STAT13,
           OUT45                    := "KAZAN1_DATA".STAT14,
           OUT46                    := "KAZAN1_TRANS_BUT_LAMBASI",
           OUT47                    := M 300.0,
           OUT48                    := "KAZAN1_DATA".STAT16,
           OUT49                    := "KAZAN1_DATA".STAT19,
           IO50                     := "KAZAN1_DATA".STAT0);
NETWORK
TITLE =
      A     "KAZAN2_DATA".STAT12;
      =     "KAZAN1_DATA".STAT2;
      L     PIW 272;
      T     "KAZAN1_DATA".STAT4;
      L     PIW 274;
      T     "KAZAN1_DATA".STAT15;
      L     "KAZAN2_DATA".STAT11;
      T     "KAZAN1_DATA".STAT6;
      O     "JEN1_DATA".STAT14;
      O     "JEN2_DATA".STAT14;
      =     "KAZAN1_DATA".STAT1;
      A     "KAZAN2_DATA".STAT16;
      =     "KAZAN1_DATA".STAT17;
      A     "KAZAN2_DATA".STAT9;
      =     "KAZAN1_DATA".STAT18;
END_FUNCTION_BLOCK

FUNCTION_BLOCK "KAZAN_2_KONTROL"	// FB 95
VERSION : 0.1
BEGIN
NETWORK
TITLE =
      CALL  "Int_To_S5Time" (
           Saat                     := "HMI_DATA".Otoklav_2_TimeData.Hours,
           Dakika                   := "HMI_DATA".Otoklav_2_TimeData.Minutes,
           HesaplananSure_S5TIME    := "KAZAN2_DATA".STAT3);
      CALL  "KAZAN_ORTAK" , DB 230 (
           IN0                      := "KAZAN2_ACIL_STOP",
           IN1                      := "KAZAN2_START",
           IN2                      := "KAZAN2_TRANSFER",
           IN3                      := "KAZAN2_BOSALTIM",
           IN4                      := "KAZAN2_KAPAK_SW",
           IN7                      := "KAZAN2_DATA".STAT1,
           IN8                      := "KAZAN2_DATA".STAT2,
           IN9                      := "KAZAN2_DATA".STAT3,
           IN10                     := "KAZAN2_DATA".STAT4,
           IN11                     := "KAZAN2_DATA".STAT5,
           IN12                     := "KAZAN2_DATA".STAT6,
           IN13                     := "500ms_delay_kazan_2",
           IN14                     := "1ms_delay_kazan_2",
           IN15                     := "kazan_2_pisirme_delay",
           IN16                     := "kazan_2_500ms_delay",
           IN17                     := "kazan_2_7s_delay",
           IN18                     := 1.000000e+01,
           IN19                     := 0.000000e+00,
           IN20                     := 2.000000e+02,
           IN21                     := 0.000000e+00,
           IN22                     := "KAZAN2_DATA".STAT15,
           IN23                     := "KAZAN2_DATA".STAT17,
           IN24                     := "KAZAN2_DATA".STAT18,
           IN27                     := "ORTAK_DATA".STAT4,
           IN29                     := "OTO_2_DELAY_BITIS",
           IN30                     := "DELAY_ADIM5_BEKLE2",
           IN31                     := T 60,
           IN32                     := T 62,
           OUT33                    := "KAZAN2_YESIL_LAMBA",
           OUT34                    := "KAZAN2_KIRMIZI_LAMBA",
           OUT35                    := "KAZAN2_DUDUK",
           OUT36                    := "KAZAN2_BOSALTIM_VALFI",
           OUT37                    := "KAZAN2_DATA".STAT7,
           OUT38                    := "KAZAN2_DATA".STAT8,
           OUT39                    := "KAZAN2_DATA".STAT9,
           OUT40                    := "KAZAN2_DATA".STAT10,
           OUT41                    := "KAZAN2_DATA".STAT11,
           OUT42                    := "KAZAN2_EMN_VALFI_BOS",
           OUT43                    := "KAZAN2_DATA".STAT12,
           OUT44                    := "KAZAN2_DATA".STAT13,
           OUT45                    := "KAZAN2_DATA".STAT14,
           OUT46                    := "KAZAN2_TRANS_BUT_LAMBASI",
           OUT47                    := M 300.1,
           OUT48                    := "KAZAN2_DATA".STAT16,
           OUT49                    := "KAZAN2_DATA".STAT19,
           IO50                     := "KAZAN2_DATA".STAT0);
NETWORK
TITLE =
      A     "KAZAN1_DATA".STAT12;
      =     "KAZAN2_DATA".STAT2;
      L     PIW 276;
      T     "KAZAN2_DATA".STAT4;
      L     PIW 278;
      T     "KAZAN2_DATA".STAT15;
      L     "KAZAN1_DATA".STAT11;
      T     "KAZAN2_DATA".STAT6;
      O     "JEN1_DATA".STAT14;
      O     "JEN2_DATA".STAT14;
      =     "KAZAN2_DATA".STAT1;
      A     "KAZAN1_DATA".STAT16;
      =     "KAZAN2_DATA".STAT17;
      A     "KAZAN1_DATA".STAT9;
      =     "KAZAN2_DATA".STAT18;
END_FUNCTION_BLOCK

FUNCTION_BLOCK "JEN1_KONTROL_BLOGU"	// FB 98
VERSION : 0.1
VAR
  STAT0 : BOOL ;
  STAT1 : BOOL ;
  STAT2 : BOOL ;
  STAT3 : BOOL ;
  STAT4 : BOOL ;
END_VAR
VAR_TEMP
  TEMP5 : BOOL ;
  TEMP6 : BOOL ;
  TEMP7 : BOOL ;
  TEMP8 : BOOL ;
  TEMP9 : BOOL ;
  TEMP10 : BOOL ;
  TEMP11 : BOOL ;
  TEMP12 : BOOL ;
  TEMP13 : BOOL ;
  TEMP14 : BOOL ;
  TEMP15 : BOOL ;
  TEMP16 : BOOL ;
END_VAR
BEGIN
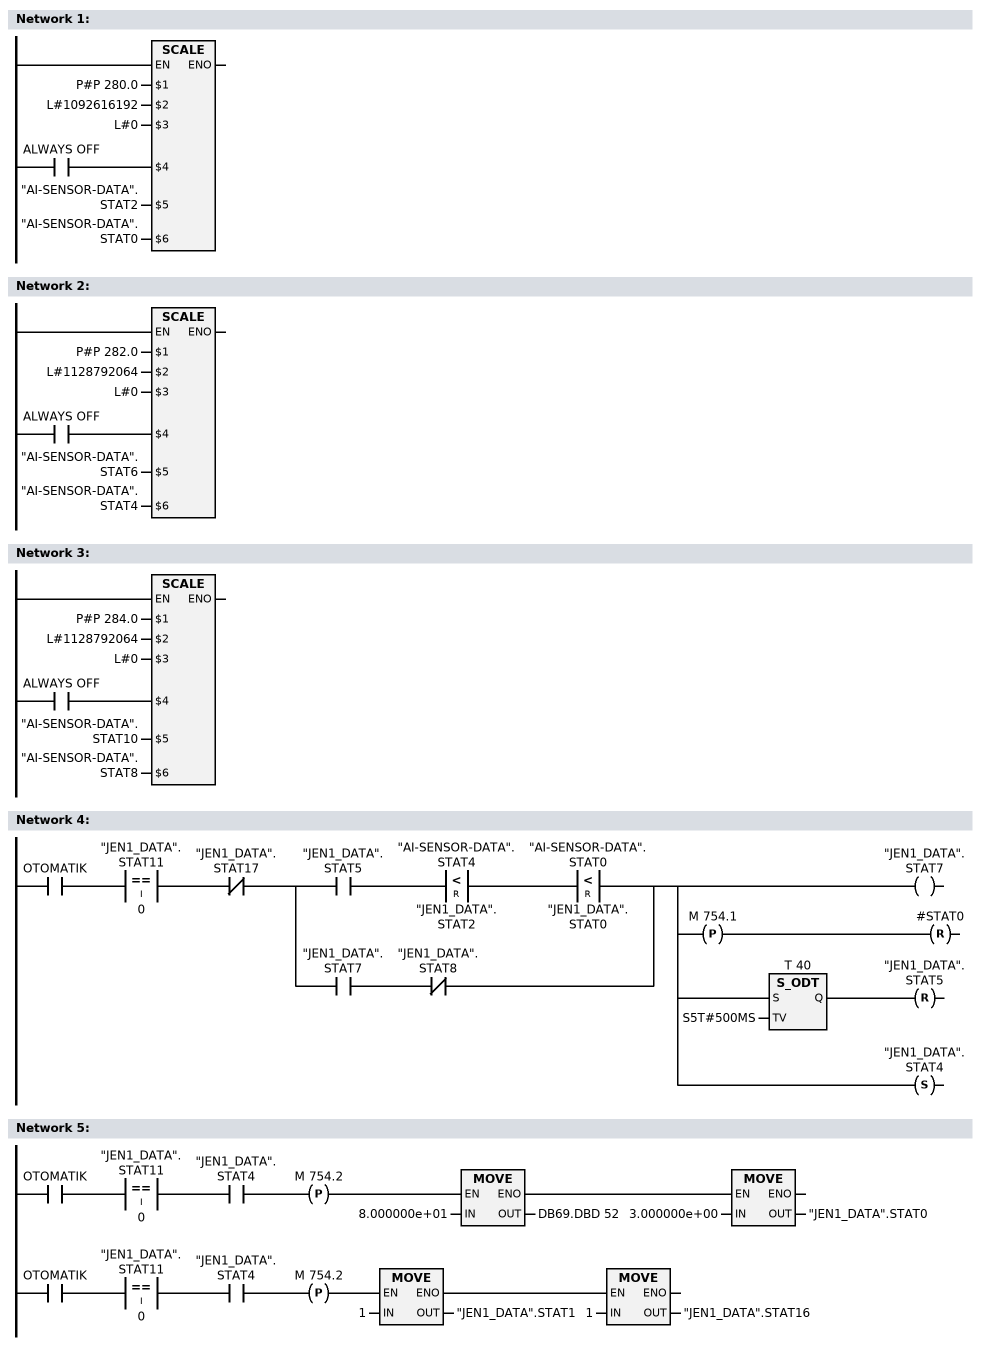
NETWORK
TITLE =
      A     "ALWAYS OFF";
      =     L 2.0;
      BLD   103;
      CALL  "SCALE" (
           $1                       := P#P 280.0,
           $2                       := L#1092616192,
           $3                       := L#0,
           $4                       := L 2.0,
           $5                       := "AI-SENSOR-DATA".STAT2,
           $6                       := "AI-SENSOR-DATA".STAT0);
      NOP   0;
NETWORK
TITLE =
      A     "ALWAYS OFF";
      =     L 2.0;
      BLD   103;
      CALL  "SCALE" (
           $1                       := P#P 282.0,
           $2                       := L#1128792064,
           $3                       := L#0,
           $4                       := L 2.0,
           $5                       := "AI-SENSOR-DATA".STAT6,
           $6                       := "AI-SENSOR-DATA".STAT4);
      NOP   0;
NETWORK
TITLE =
      A     "ALWAYS OFF";
      =     L 2.0;
      BLD   103;
      CALL  "SCALE" (
           $1                       := P#P 284.0,
           $2                       := L#1128792064,
           $3                       := L#0,
           $4                       := L 2.0,
           $5                       := "AI-SENSOR-DATA".STAT10,
           $6                       := "AI-SENSOR-DATA".STAT8);
      NOP   0;
NETWORK
TITLE =
      A     "OTOMATIK";
      A(;
      L     "JEN1_DATA".STAT11;
      L     0;
      ==I;
      );
      AN    "JEN1_DATA".STAT17;
      A(;
      A     "JEN1_DATA".STAT5;
      A(;
      L     "AI-SENSOR-DATA".STAT4;
      L     "JEN1_DATA".STAT2;
      <R;
      );
      A(;
      L     "AI-SENSOR-DATA".STAT0;
      L     "JEN1_DATA".STAT0;
      <R;
      );
      O;
      A     "JEN1_DATA".STAT7;
      AN    "JEN1_DATA".STAT8;
      );
      =     L 2.0;
      A     L 2.0;
      BLD   102;
      =     "JEN1_DATA".STAT7;
      A     L 2.0;
      FP    M 754.1;
      R     #STAT0;
      A     L 2.0;
      L     S5T#500MS;
      SD    T 40;
      NOP   0;
      NOP   0;
      NOP   0;
      A     T 40;
      R     "JEN1_DATA".STAT5;
      A     L 2.0;
      BLD   102;
      S     "JEN1_DATA".STAT4;
NETWORK
TITLE =
      A     "OTOMATIK";
      A(;
      L     "JEN1_DATA".STAT11;
      L     0;
      ==I;
      );
      A     "JEN1_DATA".STAT4;
      FP    M 754.2;
      =     L 2.0;
      A(;
      A     L 2.0;
      JNB   _001;
      L     8.000000e+01;
      T     DB69.DBD 52;
      SET;
      SAVE;
      CLR;
_001: A     BR;
      );
      JNB   _002;
      L     3.000000e+00;
      T     "JEN1_DATA".STAT0;
_002: NOP   0;
      A(;
      A     L 2.0;
      JNB   _003;
      L     1;
      T     "JEN1_DATA".STAT1;
      SET;
      SAVE;
      CLR;
_003: A     BR;
      );
      JNB   _004;
      L     1;
      T     "JEN1_DATA".STAT16;
_004: NOP   0;
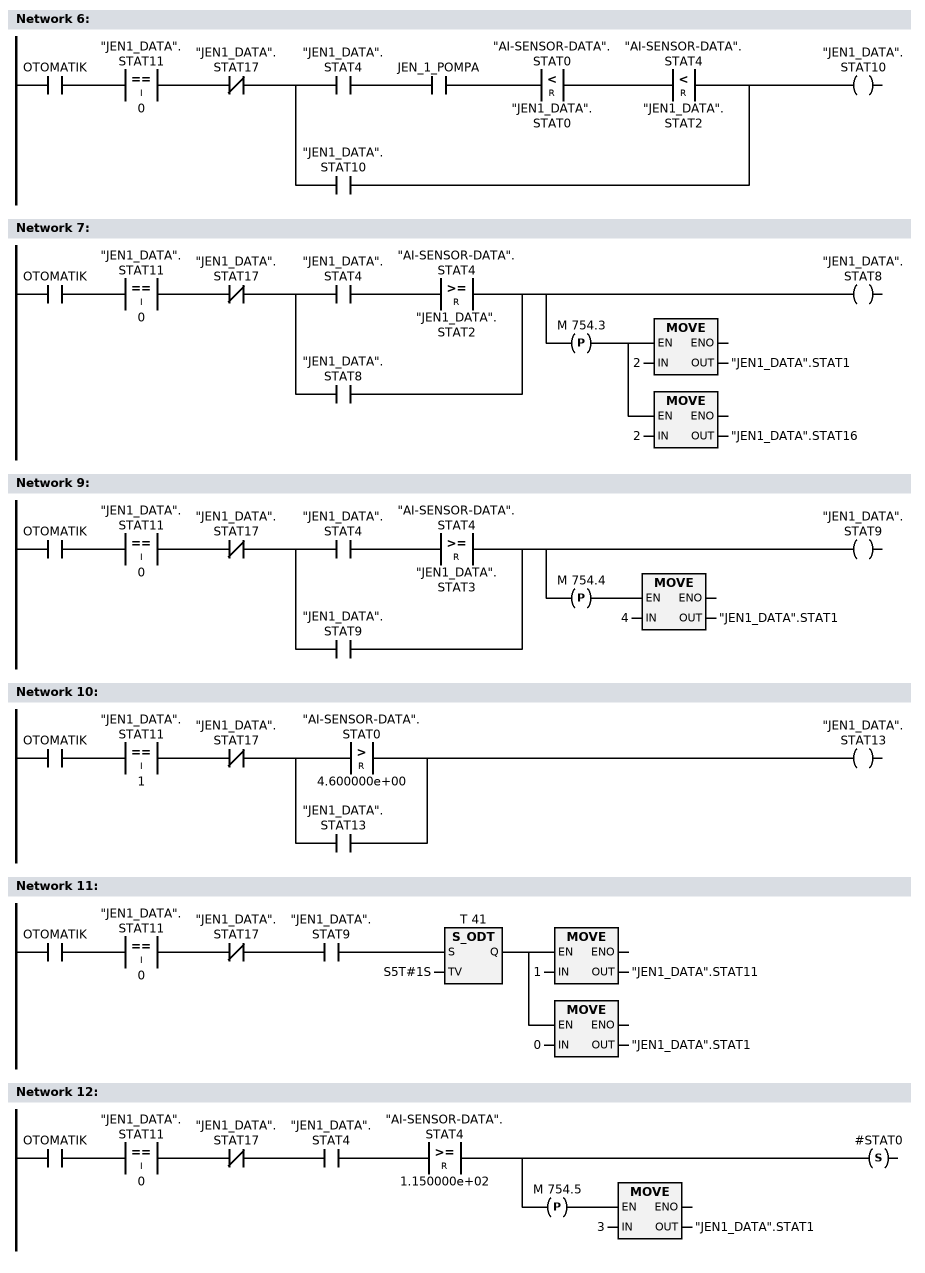
NETWORK
TITLE =
      A     "OTOMATIK";
      A(;
      L     "JEN1_DATA".STAT11;
      L     0;
      ==I;
      );
      AN    "JEN1_DATA".STAT17;
      A(;
      A     "JEN1_DATA".STAT4;
      A     "JEN_1_POMPA";
      A(;
      L     "AI-SENSOR-DATA".STAT0;
      L     "JEN1_DATA".STAT0;
      <R;
      );
      A(;
      L     "AI-SENSOR-DATA".STAT4;
      L     "JEN1_DATA".STAT2;
      <R;
      );
      O     "JEN1_DATA".STAT10;
      );
      =     "JEN1_DATA".STAT10;
NETWORK
TITLE =
      A     "OTOMATIK";
      A(;
      L     "JEN1_DATA".STAT11;
      L     0;
      ==I;
      );
      AN    "JEN1_DATA".STAT17;
      A(;
      A     "JEN1_DATA".STAT4;
      A(;
      L     "AI-SENSOR-DATA".STAT4;
      L     "JEN1_DATA".STAT2;
      >=R;
      );
      O     "JEN1_DATA".STAT8;
      );
      =     L 2.0;
      A     L 2.0;
      BLD   102;
      =     "JEN1_DATA".STAT8;
      A     L 2.0;
      FP    M 754.3;
      =     L 2.1;
      A     L 2.1;
      JNB   _005;
      L     2;
      T     "JEN1_DATA".STAT1;
_005: NOP   0;
      A     L 2.1;
      JNB   _006;
      L     2;
      T     "JEN1_DATA".STAT16;
_006: NOP   0;
NETWORK
TITLE =
      A(;
      A     "JEN1_DATA".STAT8;
      FP    "SET2_ULASMADI_RIS";
      S     "SET2_ULASMADI_SR";
      A(;
      O(;
      L     "JEN1_DATA".STAT11;
      L     1;
      ==I;
      );
      O     "JEN1_DATA".STAT17;
      );
      R     "SET2_ULASMADI_SR";
      A     "SET2_ULASMADI_SR";
      );
      L     S5T#1M30S;
      SD    "TIM_SET2_ULASMADI";
      NOP   0;
      NOP   0;
      NOP   0;
      A     "TIM_SET2_ULASMADI";
      =     "JEN1_DATA".STAT22;
NETWORK
TITLE =
      A     "OTOMATIK";
      A(;
      L     "JEN1_DATA".STAT11;
      L     0;
      ==I;
      );
      AN    "JEN1_DATA".STAT17;
      A(;
      A     "JEN1_DATA".STAT4;
      A(;
      L     "AI-SENSOR-DATA".STAT4;
      L     "JEN1_DATA".STAT3;
      >=R;
      );
      O     "JEN1_DATA".STAT9;
      );
      =     L 2.0;
      A     L 2.0;
      BLD   102;
      =     "JEN1_DATA".STAT9;
      A     L 2.0;
      FP    M 754.4;
      JNB   _007;
      L     4;
      T     "JEN1_DATA".STAT1;
_007: NOP   0;
NETWORK
TITLE =
      A     "OTOMATIK";
      A(;
      L     "JEN1_DATA".STAT11;
      L     1;
      ==I;
      );
      AN    "JEN1_DATA".STAT17;
      A(;
      O(;
      L     "AI-SENSOR-DATA".STAT0;
      L     4.600000e+00;
      >R;
      );
      O     "JEN1_DATA".STAT13;
      );
      =     "JEN1_DATA".STAT13;
NETWORK
TITLE =
      A     "OTOMATIK";
      A(;
      L     "JEN1_DATA".STAT11;
      L     0;
      ==I;
      );
      AN    "JEN1_DATA".STAT17;
      A     "JEN1_DATA".STAT9;
      L     S5T#1S;
      SD    T 41;
      NOP   0;
      NOP   0;
      NOP   0;
      A     T 41;
      =     L 2.0;
      A     L 2.0;
      JNB   _008;
      L     1;
      T     "JEN1_DATA".STAT11;
_008: NOP   0;
      A     L 2.0;
      JNB   _009;
      L     0;
      T     "JEN1_DATA".STAT1;
_009: NOP   0;
NETWORK
TITLE =
      A     "OTOMATIK";
      A(;
      L     "JEN1_DATA".STAT11;
      L     0;
      ==I;
      );
      AN    "JEN1_DATA".STAT17;
      A     "JEN1_DATA".STAT4;
      A(;
      L     "AI-SENSOR-DATA".STAT4;
      L     1.150000e+02;
      >=R;
      );
      =     L 2.0;
      A     L 2.0;
      BLD   102;
      S     #STAT0;
      A     L 2.0;
      FP    M 754.5;
      JNB   _00a;
      L     3;
      T     "JEN1_DATA".STAT1;
_00a: NOP   0;
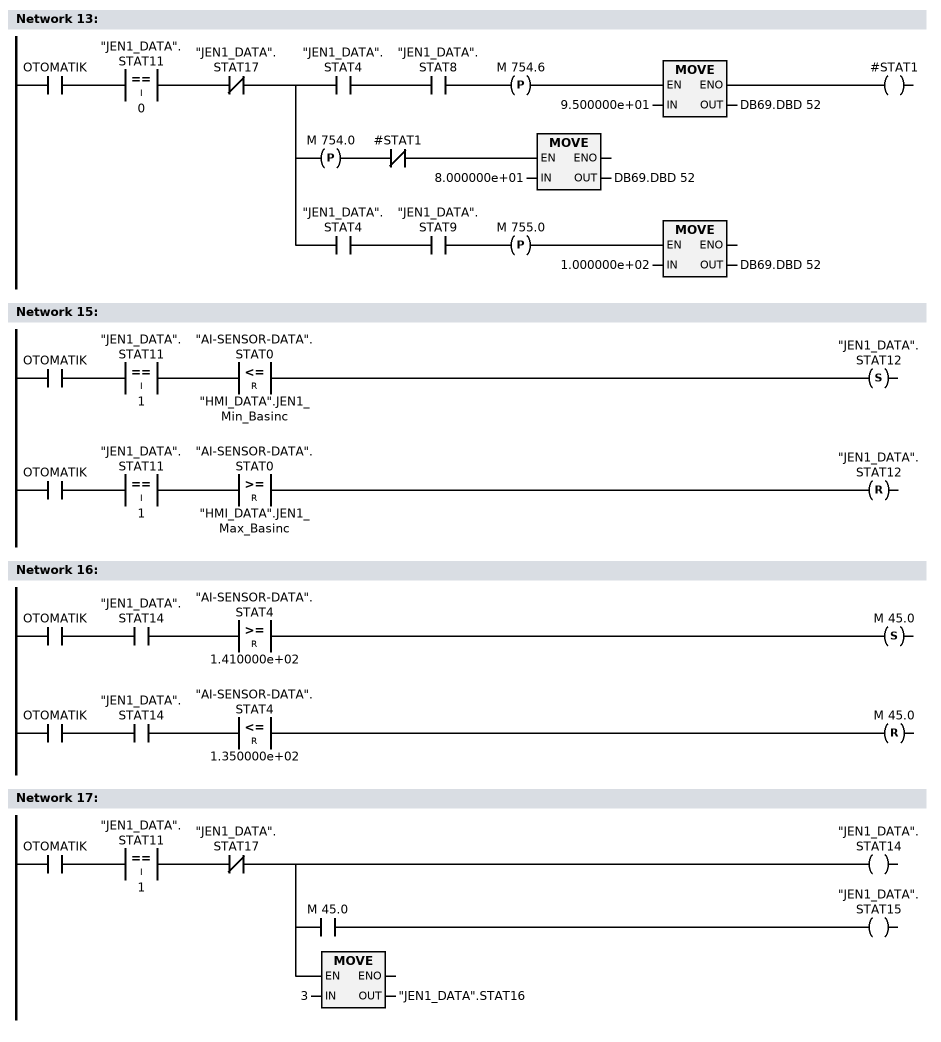
NETWORK
TITLE =
      A     "OTOMATIK";
      A(;
      L     "JEN1_DATA".STAT11;
      L     0;
      ==I;
      );
      AN    "JEN1_DATA".STAT17;
      =     L 2.0;
      A     L 2.0;
      A     "JEN1_DATA".STAT4;
      A     "JEN1_DATA".STAT8;
      FP    M 754.6;
      JNB   _00b;
      L     9.500000e+01;
      T     DB69.DBD 52;
      SET;
      SAVE;
      CLR;
_00b: A     BR;
      =     #STAT1;
      A     L 2.0;
      FP    M 754.0;
      AN    #STAT1;
      JNB   _00c;
      L     8.000000e+01;
      T     DB69.DBD 52;
_00c: NOP   0;
      A     L 2.0;
      A     "JEN1_DATA".STAT4;
      A     "JEN1_DATA".STAT9;
      FP    M 755.0;
      JNB   _00d;
      L     1.000000e+02;
      T     DB69.DBD 52;
_00d: NOP   0;
NETWORK
TITLE =
NETWORK
TITLE =
      A     "OTOMATIK";
      A(;
      L     "JEN1_DATA".STAT11;
      L     1;
      ==I;
      );
      A(;
      L     "AI-SENSOR-DATA".STAT0;
      L     "HMI_DATA".JEN1_Min_Basinc;
      <=R;
      );
      S     "JEN1_DATA".STAT12;
      A     "OTOMATIK";
      A(;
      L     "JEN1_DATA".STAT11;
      L     1;
      ==I;
      );
      A(;
      L     "AI-SENSOR-DATA".STAT0;
      L     "HMI_DATA".JEN1_Max_Basinc;
      >=R;
      );
      R     "JEN1_DATA".STAT12;
      NOP   0;
NETWORK
TITLE =
      A     "OTOMATIK";
      A     "JEN1_DATA".STAT14;
      A(;
      L     "AI-SENSOR-DATA".STAT4;
      L     1.410000e+02;
      >=R;
      );
      S     M 45.0;
      A     "OTOMATIK";
      A     "JEN1_DATA".STAT14;
      A(;
      L     "AI-SENSOR-DATA".STAT4;
      L     1.350000e+02;
      <=R;
      );
      R     M 45.0;
      NOP   0;
NETWORK
TITLE =
      A     "OTOMATIK";
      A(;
      L     "JEN1_DATA".STAT11;
      L     1;
      ==I;
      );
      AN    "JEN1_DATA".STAT17;
      =     L 2.0;
      A     L 2.0;
      BLD   102;
      =     "JEN1_DATA".STAT14;
      A     L 2.0;
      A     M 45.0;
      =     "JEN1_DATA".STAT15;
      A     L 2.0;
      JNB   _00e;
      L     3;
      T     "JEN1_DATA".STAT16;
_00e: NOP   0;
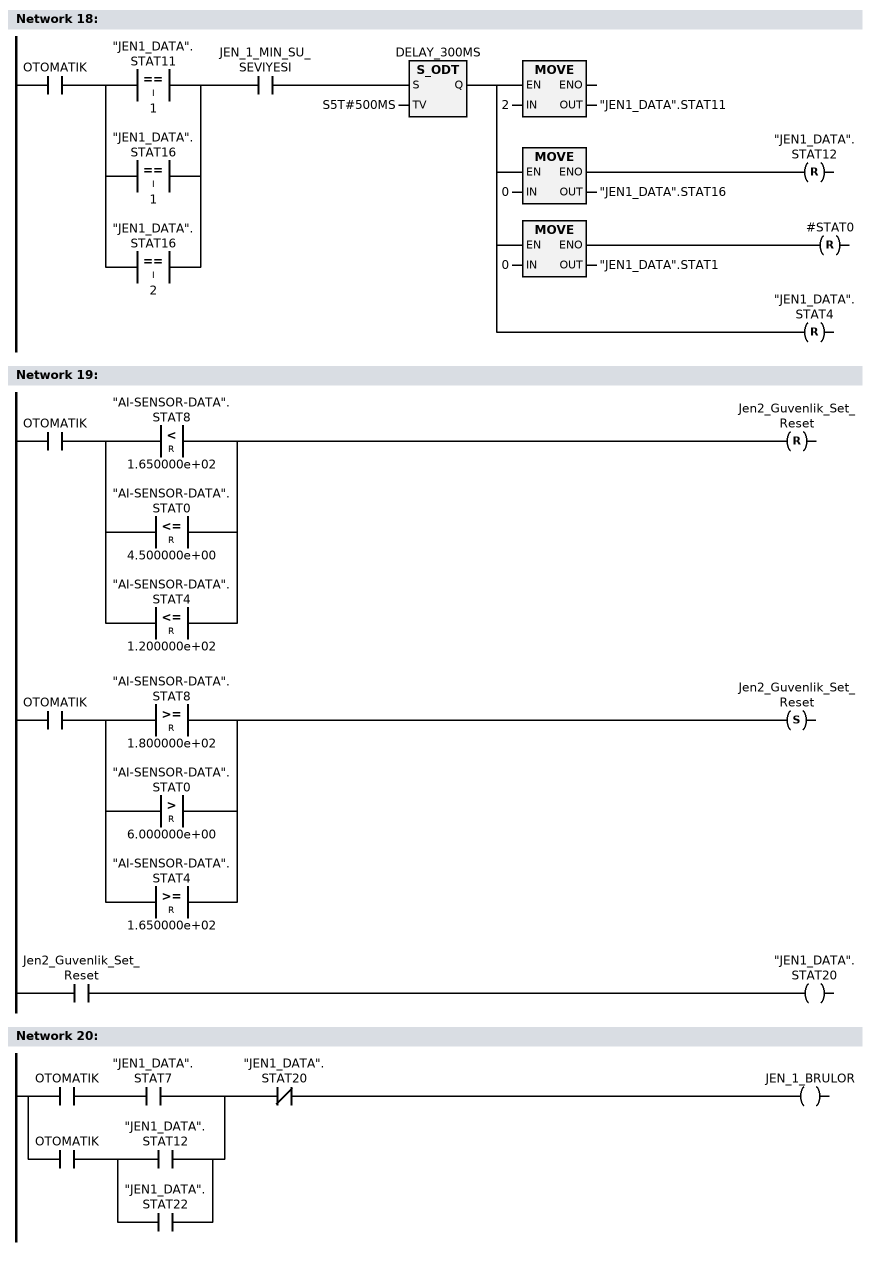
NETWORK
TITLE =
      A     "OTOMATIK";
      A(;
      O(;
      L     "JEN1_DATA".STAT11;
      L     1;
      ==I;
      );
      O(;
      L     "JEN1_DATA".STAT16;
      L     1;
      ==I;
      );
      O(;
      L     "JEN1_DATA".STAT16;
      L     2;
      ==I;
      );
      );
      A     "JEN_1_MIN_SU_SEVIYESI";
      L     S5T#500MS;
      SD    "DELAY_300MS";
      NOP   0;
      NOP   0;
      NOP   0;
      A     "DELAY_300MS";
      =     L 2.0;
      A     L 2.0;
      JNB   _00f;
      L     2;
      T     "JEN1_DATA".STAT11;
_00f: NOP   0;
      A     L 2.0;
      JNB   _010;
      L     0;
      T     "JEN1_DATA".STAT16;
      SET;
      SAVE;
      CLR;
_010: A     BR;
      R     "JEN1_DATA".STAT12;
      A     L 2.0;
      JNB   _011;
      L     0;
      T     "JEN1_DATA".STAT1;
      SET;
      SAVE;
      CLR;
_011: A     BR;
      R     #STAT0;
      A     L 2.0;
      BLD   102;
      R     "JEN1_DATA".STAT4;
NETWORK
TITLE =
      A     "OTOMATIK";
      A(;
      O(;
      L     "AI-SENSOR-DATA".STAT8;
      L     1.650000e+02;
      <R;
      );
      O(;
      L     "AI-SENSOR-DATA".STAT0;
      L     4.500000e+00;
      <=R;
      );
      O(;
      L     "AI-SENSOR-DATA".STAT4;
      L     1.200000e+02;
      <=R;
      );
      );
      R     "Jen2_Guvenlik_Set_Reset";
      A     "OTOMATIK";
      A(;
      O(;
      L     "AI-SENSOR-DATA".STAT8;
      L     1.800000e+02;
      >=R;
      );
      O(;
      L     "AI-SENSOR-DATA".STAT0;
      L     6.000000e+00;
      >R;
      );
      O(;
      L     "AI-SENSOR-DATA".STAT4;
      L     1.650000e+02;
      >=R;
      );
      );
      S     "Jen2_Guvenlik_Set_Reset";
      A     "Jen2_Guvenlik_Set_Reset";
      =     "JEN1_DATA".STAT20;
NETWORK
TITLE =
      A(;
      A     "OTOMATIK";
      A     "JEN1_DATA".STAT7;
      O;
      A     "OTOMATIK";
      A(;
      O     "JEN1_DATA".STAT12;
      O     "JEN1_DATA".STAT22;
      );
      );
      AN    "JEN1_DATA".STAT20;
      =     "JEN_1_BRULOR";
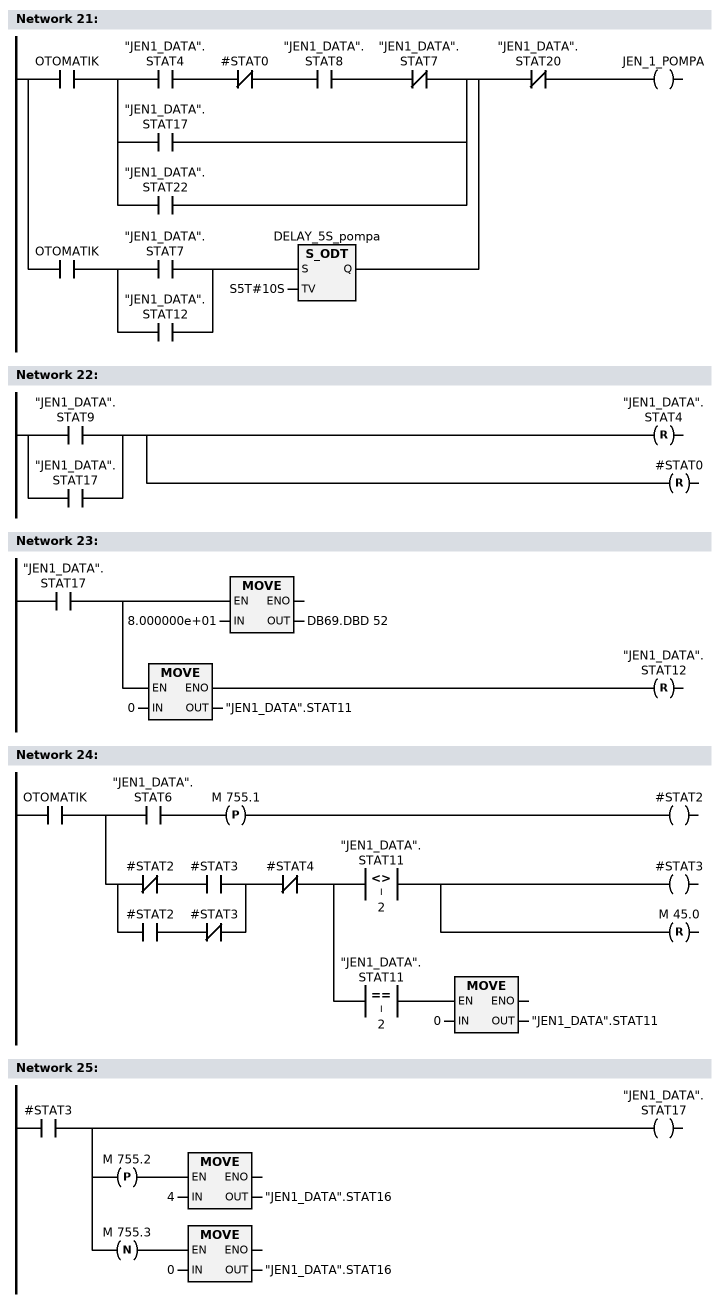
NETWORK
TITLE =
      A(;
      A     "OTOMATIK";
      A(;
      A     "JEN1_DATA".STAT4;
      AN    #STAT0;
      A     "JEN1_DATA".STAT8;
      AN    "JEN1_DATA".STAT7;
      O     "JEN1_DATA".STAT17;
      O     "JEN1_DATA".STAT22;
      );
      O(;
      A     "OTOMATIK";
      A(;
      O     "JEN1_DATA".STAT7;
      O     "JEN1_DATA".STAT12;
      );
      L     S5T#10S;
      SD    "DELAY_5S_pompa";
      NOP   0;
      NOP   0;
      NOP   0;
      A     "DELAY_5S_pompa";
      );
      );
      AN    "JEN1_DATA".STAT20;
      =     "JEN_1_POMPA";
NETWORK
TITLE =
      O     "JEN1_DATA".STAT9;
      O     "JEN1_DATA".STAT17;
      R     "JEN1_DATA".STAT4;
      R     #STAT0;
NETWORK
TITLE =
      A     "JEN1_DATA".STAT17;
      =     L 2.0;
      A     L 2.0;
      JNB   _012;
      L     8.000000e+01;
      T     DB69.DBD 52;
_012: NOP   0;
      A     L 2.0;
      JNB   _013;
      L     0;
      T     "JEN1_DATA".STAT11;
      SET;
      SAVE;
      CLR;
_013: A     BR;
      R     "JEN1_DATA".STAT12;
NETWORK
TITLE =
      A     "OTOMATIK";
      =     L 2.0;
      A     L 2.0;
      A     "JEN1_DATA".STAT6;
      FP    M 755.1;
      =     #STAT2;
      A     L 2.0;
      A(;
      AN    #STAT2;
      A     #STAT3;
      O;
      A     #STAT2;
      AN    #STAT3;
      );
      AN    #STAT4;
      =     L 2.1;
      A     L 2.1;
      A(;
      L     "JEN1_DATA".STAT11;
      L     2;
      <>I;
      );
      =     #STAT3;
      R     M 45.0;
      A     L 2.1;
      A(;
      L     "JEN1_DATA".STAT11;
      L     2;
      ==I;
      );
      JNB   _014;
      L     0;
      T     "JEN1_DATA".STAT11;
_014: NOP   0;
NETWORK
TITLE =
      A     #STAT3;
      =     L 2.0;
      A     L 2.0;
      BLD   102;
      =     "JEN1_DATA".STAT17;
      A     L 2.0;
      FP    M 755.2;
      JNB   _015;
      L     4;
      T     "JEN1_DATA".STAT16;
_015: NOP   0;
      A     L 2.0;
      FN    M 755.3;
      JNB   _016;
      L     0;
      T     "JEN1_DATA".STAT16;
_016: NOP   0;
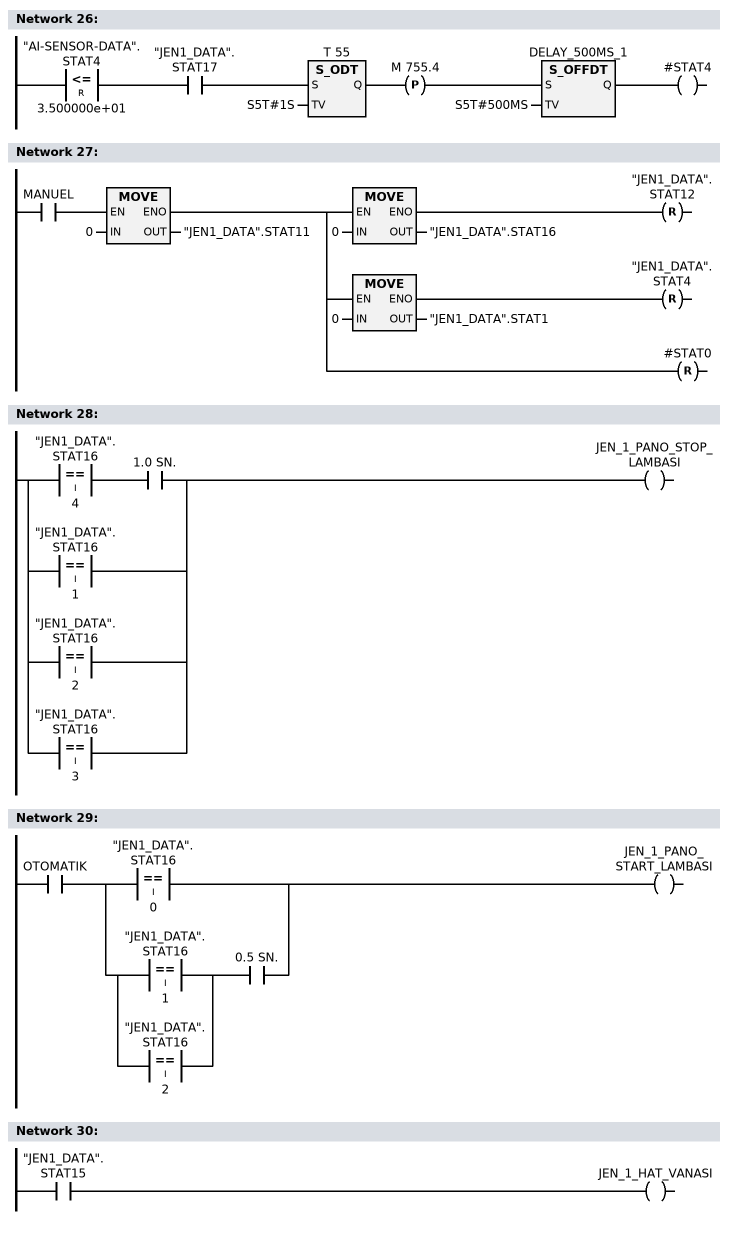
NETWORK
TITLE =
      A(;
      A(;
      L     "AI-SENSOR-DATA".STAT4;
      L     3.500000e+01;
      <=R;
      );
      A     "JEN1_DATA".STAT17;
      L     S5T#1S;
      SD    T 55;
      NOP   0;
      NOP   0;
      NOP   0;
      A     T 55;
      );
      FP    M 755.4;
      L     S5T#500MS;
      SF    "DELAY_500MS_1";
      NOP   0;
      NOP   0;
      NOP   0;
      A     "DELAY_500MS_1";
      =     #STAT4;
NETWORK
TITLE =
      A     "MANUEL";
      JNB   _017;
      L     0;
      T     "JEN1_DATA".STAT11;
      SET;
      SAVE;
      CLR;
_017: A     BR;
      =     L 2.0;
      A     L 2.0;
      JNB   _018;
      L     0;
      T     "JEN1_DATA".STAT16;
      SET;
      SAVE;
      CLR;
_018: A     BR;
      R     "JEN1_DATA".STAT12;
      A     L 2.0;
      JNB   _019;
      L     0;
      T     "JEN1_DATA".STAT1;
      SET;
      SAVE;
      CLR;
_019: A     BR;
      R     "JEN1_DATA".STAT4;
      A     L 2.0;
      BLD   102;
      R     #STAT0;
NETWORK
TITLE =
      A(;
      L     "JEN1_DATA".STAT16;
      L     4;
      ==I;
      );
      A     "1.0 SN.";
      O(;
      L     "JEN1_DATA".STAT16;
      L     1;
      ==I;
      );
      O(;
      L     "JEN1_DATA".STAT16;
      L     2;
      ==I;
      );
      O(;
      L     "JEN1_DATA".STAT16;
      L     3;
      ==I;
      );
      =     "JEN_1_PANO_STOP_LAMBASI";
NETWORK
TITLE =
      A     "OTOMATIK";
      A(;
      O(;
      L     "JEN1_DATA".STAT16;
      L     0;
      ==I;
      );
      O;
      A(;
      O(;
      L     "JEN1_DATA".STAT16;
      L     1;
      ==I;
      );
      O(;
      L     "JEN1_DATA".STAT16;
      L     2;
      ==I;
      );
      );
      A     "0.5 SN.";
      );
      =     "JEN_1_PANO_START_LAMBASI";
NETWORK
TITLE =
      A     "JEN1_DATA".STAT15;
      =     "JEN_1_HAT_VANASI";
END_FUNCTION_BLOCK

FUNCTION_BLOCK "JEN2_KONTROL_BLOGU"	// FB 99
VERSION : 0.1
VAR
  STAT0 : BOOL ;
  STAT1 : BOOL ;
  STAT2 : BOOL ;
  STAT3 : BOOL ;
  STAT4 : BOOL ;
  STAT5 : BOOL ;
  STAT6 : BOOL ;
  STAT7 : BOOL ;
  STAT8 : BOOL ;
  STAT9 : BOOL ;
END_VAR
BEGIN
NETWORK
TITLE =
      A     "ALWAYS OFF";
      =     L 0.0;
      BLD   103;
      A(;
      A     "ALWAYS OFF";
      =     L 0.1;
      BLD   103;
      CALL  "SCALE" (
           $1                       := P#P 286.0,
           $2                       := L#1092616192,
           $3                       := L#0,
           $4                       := L 0.1,
           $5                       := "AI-SENSOR-DATA".STAT3,
           $6                       := "AI-SENSOR-DATA".STAT1);
      A     BR;
      );
      JNB   _001;
      CALL  "SCALE" (
           $1                       := P#P 288.0,
           $2                       := L#1128792064,
           $3                       := L#0,
           $4                       := L 0.0,
           $5                       := "AI-SENSOR-DATA".STAT7,
           $6                       := "AI-SENSOR-DATA".STAT5);
_001: NOP   0;
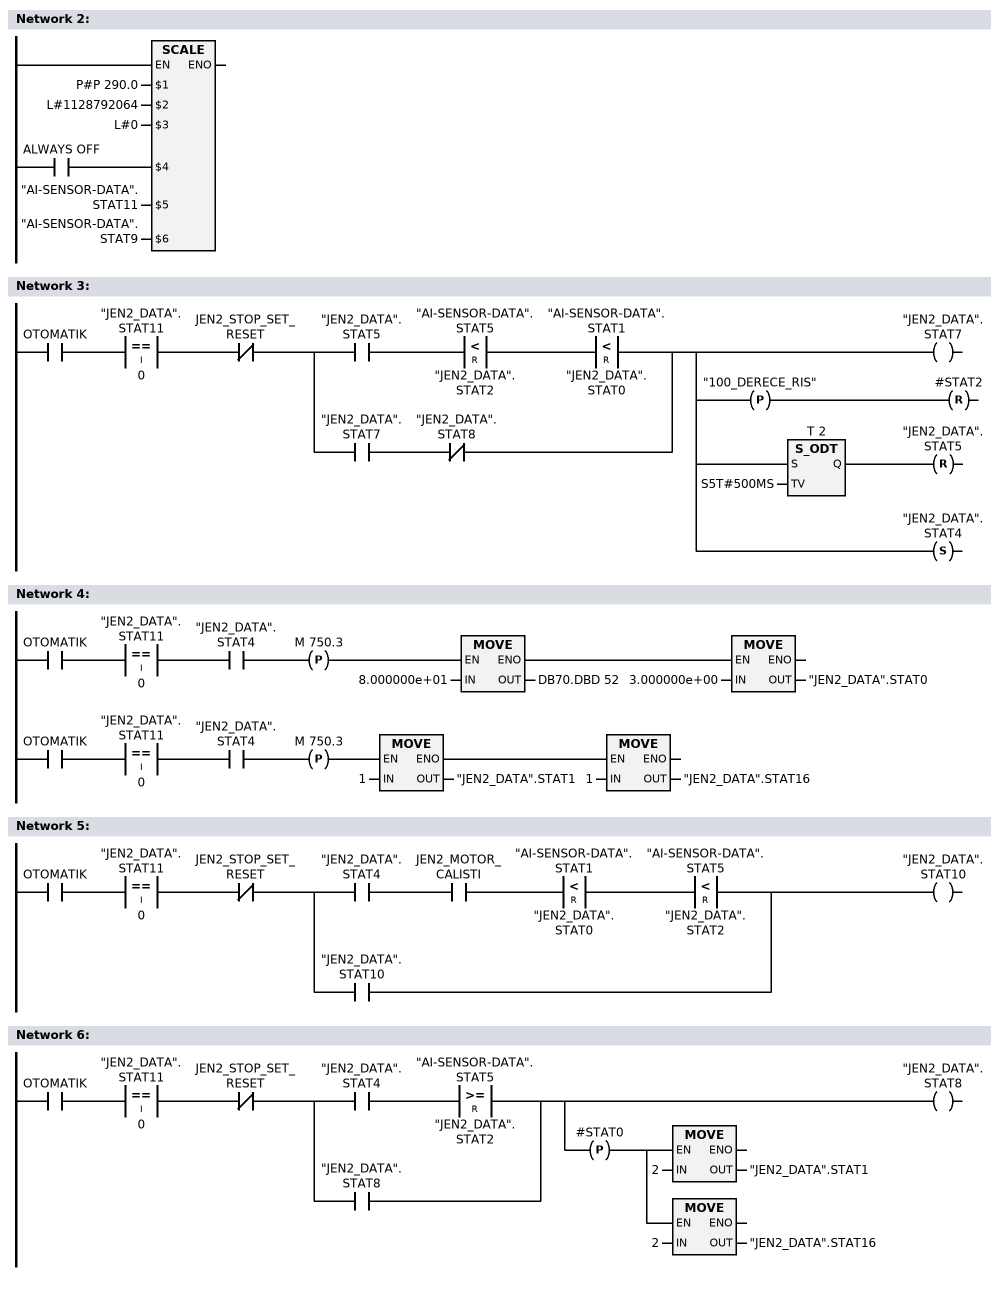
NETWORK
TITLE =
      A     "ALWAYS OFF";
      =     L 0.0;
      BLD   103;
      CALL  "SCALE" (
           $1                       := P#P 290.0,
           $2                       := L#1128792064,
           $3                       := L#0,
           $4                       := L 0.0,
           $5                       := "AI-SENSOR-DATA".STAT11,
           $6                       := "AI-SENSOR-DATA".STAT9);
      NOP   0;
NETWORK
TITLE =
      A     "OTOMATIK";
      A(;
      L     "JEN2_DATA".STAT11;
      L     0;
      ==I;
      );
      AN    "JEN2_STOP_SET_RESET";
      A(;
      A     "JEN2_DATA".STAT5;
      A(;
      L     "AI-SENSOR-DATA".STAT5;
      L     "JEN2_DATA".STAT2;
      <R;
      );
      A(;
      L     "AI-SENSOR-DATA".STAT1;
      L     "JEN2_DATA".STAT0;
      <R;
      );
      O;
      A     "JEN2_DATA".STAT7;
      AN    "JEN2_DATA".STAT8;
      );
      =     L 0.0;
      A     L 0.0;
      BLD   102;
      =     "JEN2_DATA".STAT7;
      A     L 0.0;
      FP    "100_DERECE_RIS";
      R     #STAT2;
      A     L 0.0;
      L     S5T#500MS;
      SD    T 2;
      NOP   0;
      NOP   0;
      NOP   0;
      A     T 2;
      R     "JEN2_DATA".STAT5;
      A     L 0.0;
      BLD   102;
      S     "JEN2_DATA".STAT4;
NETWORK
TITLE =
      A     "OTOMATIK";
      A(;
      L     "JEN2_DATA".STAT11;
      L     0;
      ==I;
      );
      A     "JEN2_DATA".STAT4;
      FP    M 750.3;
      =     L 0.0;
      A(;
      A     L 0.0;
      JNB   _002;
      L     8.000000e+01;
      T     DB70.DBD 52;
      SET;
      SAVE;
      CLR;
_002: A     BR;
      );
      JNB   _003;
      L     3.000000e+00;
      T     "JEN2_DATA".STAT0;
_003: NOP   0;
      A(;
      A     L 0.0;
      JNB   _004;
      L     1;
      T     "JEN2_DATA".STAT1;
      SET;
      SAVE;
      CLR;
_004: A     BR;
      );
      JNB   _005;
      L     1;
      T     "JEN2_DATA".STAT16;
_005: NOP   0;
NETWORK
TITLE =
      A     "OTOMATIK";
      A(;
      L     "JEN2_DATA".STAT11;
      L     0;
      ==I;
      );
      AN    "JEN2_STOP_SET_RESET";
      A(;
      A     "JEN2_DATA".STAT4;
      A     "JEN2_MOTOR_CALISTI";
      A(;
      L     "AI-SENSOR-DATA".STAT1;
      L     "JEN2_DATA".STAT0;
      <R;
      );
      A(;
      L     "AI-SENSOR-DATA".STAT5;
      L     "JEN2_DATA".STAT2;
      <R;
      );
      O     "JEN2_DATA".STAT10;
      );
      =     "JEN2_DATA".STAT10;
NETWORK
TITLE =
      A     "OTOMATIK";
      A(;
      L     "JEN2_DATA".STAT11;
      L     0;
      ==I;
      );
      AN    "JEN2_STOP_SET_RESET";
      A(;
      A     "JEN2_DATA".STAT4;
      A(;
      L     "AI-SENSOR-DATA".STAT5;
      L     "JEN2_DATA".STAT2;
      >=R;
      );
      O     "JEN2_DATA".STAT8;
      );
      =     L 0.0;
      A     L 0.0;
      BLD   102;
      =     "JEN2_DATA".STAT8;
      A     L 0.0;
      FP    #STAT0;
      =     L 0.1;
      A     L 0.1;
      JNB   _006;
      L     2;
      T     "JEN2_DATA".STAT1;
_006: NOP   0;
      A     L 0.1;
      JNB   _007;
      L     2;
      T     "JEN2_DATA".STAT16;
_007: NOP   0;
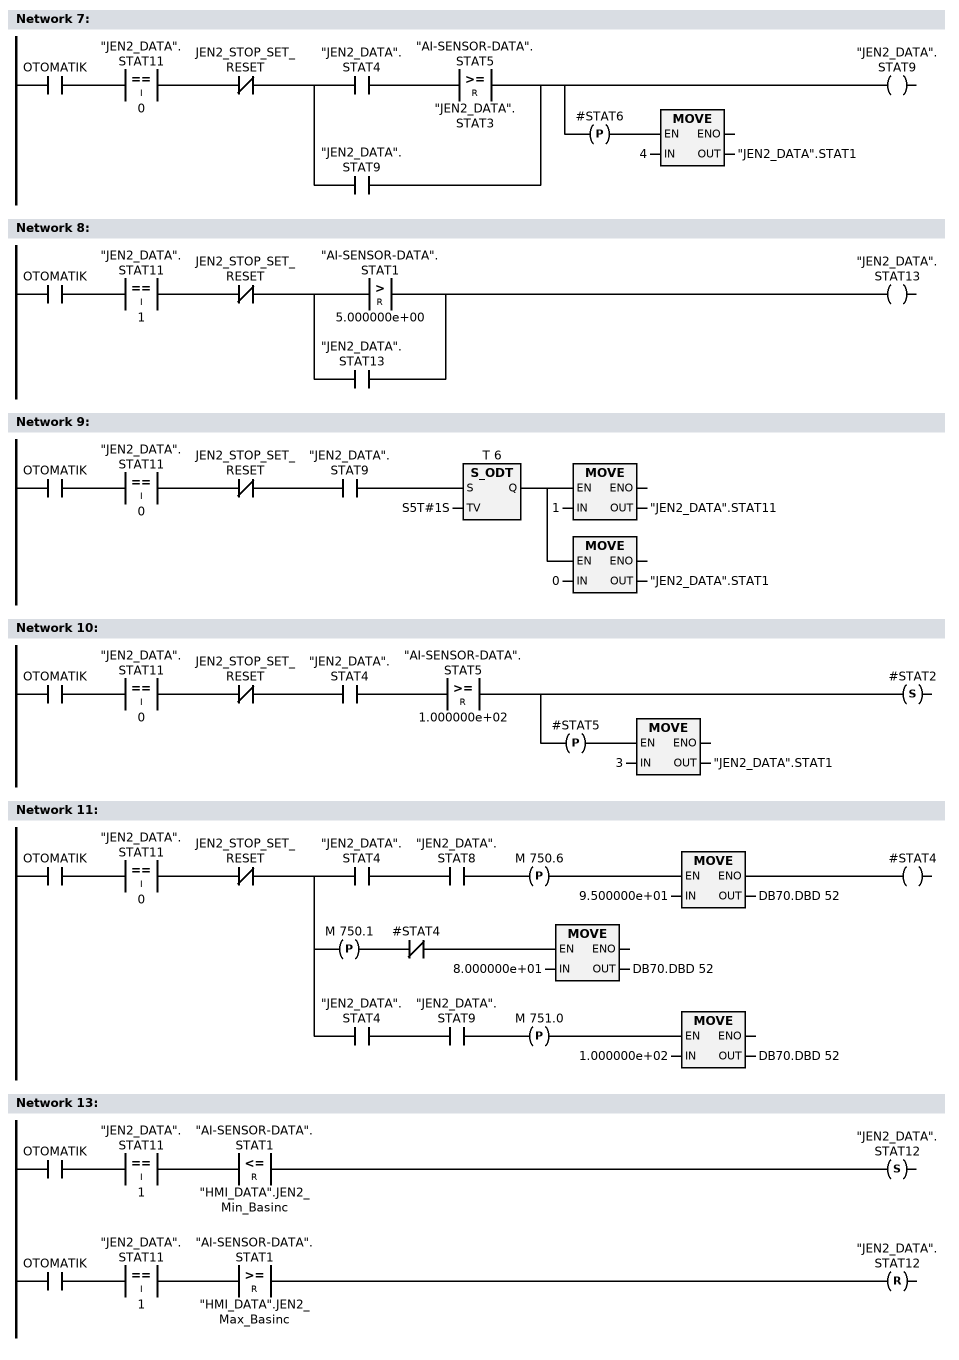
NETWORK
TITLE =
      A     "OTOMATIK";
      A(;
      L     "JEN2_DATA".STAT11;
      L     0;
      ==I;
      );
      AN    "JEN2_STOP_SET_RESET";
      A(;
      A     "JEN2_DATA".STAT4;
      A(;
      L     "AI-SENSOR-DATA".STAT5;
      L     "JEN2_DATA".STAT3;
      >=R;
      );
      O     "JEN2_DATA".STAT9;
      );
      =     L 0.0;
      A     L 0.0;
      BLD   102;
      =     "JEN2_DATA".STAT9;
      A     L 0.0;
      FP    #STAT6;
      JNB   _008;
      L     4;
      T     "JEN2_DATA".STAT1;
_008: NOP   0;
NETWORK
TITLE =
      A     "OTOMATIK";
      A(;
      L     "JEN2_DATA".STAT11;
      L     1;
      ==I;
      );
      AN    "JEN2_STOP_SET_RESET";
      A(;
      O(;
      L     "AI-SENSOR-DATA".STAT1;
      L     5.000000e+00;
      >R;
      );
      O     "JEN2_DATA".STAT13;
      );
      =     "JEN2_DATA".STAT13;
NETWORK
TITLE =
      A     "OTOMATIK";
      A(;
      L     "JEN2_DATA".STAT11;
      L     0;
      ==I;
      );
      AN    "JEN2_STOP_SET_RESET";
      A     "JEN2_DATA".STAT9;
      L     S5T#1S;
      SD    T 6;
      NOP   0;
      NOP   0;
      NOP   0;
      A     T 6;
      =     L 0.0;
      A     L 0.0;
      JNB   _009;
      L     1;
      T     "JEN2_DATA".STAT11;
_009: NOP   0;
      A     L 0.0;
      JNB   _00a;
      L     0;
      T     "JEN2_DATA".STAT1;
_00a: NOP   0;
NETWORK
TITLE =
      A     "OTOMATIK";
      A(;
      L     "JEN2_DATA".STAT11;
      L     0;
      ==I;
      );
      AN    "JEN2_STOP_SET_RESET";
      A     "JEN2_DATA".STAT4;
      A(;
      L     "AI-SENSOR-DATA".STAT5;
      L     1.000000e+02;
      >=R;
      );
      =     L 0.0;
      A     L 0.0;
      BLD   102;
      S     #STAT2;
      A     L 0.0;
      FP    #STAT5;
      JNB   _00b;
      L     3;
      T     "JEN2_DATA".STAT1;
_00b: NOP   0;
NETWORK
TITLE =
      A     "OTOMATIK";
      A(;
      L     "JEN2_DATA".STAT11;
      L     0;
      ==I;
      );
      AN    "JEN2_STOP_SET_RESET";
      =     L 0.0;
      A     L 0.0;
      A     "JEN2_DATA".STAT4;
      A     "JEN2_DATA".STAT8;
      FP    M 750.6;
      JNB   _00c;
      L     9.500000e+01;
      T     DB70.DBD 52;
      SET;
      SAVE;
      CLR;
_00c: A     BR;
      =     #STAT4;
      A     L 0.0;
      FP    M 750.1;
      AN    #STAT4;
      JNB   _00d;
      L     8.000000e+01;
      T     DB70.DBD 52;
_00d: NOP   0;
      A     L 0.0;
      A     "JEN2_DATA".STAT4;
      A     "JEN2_DATA".STAT9;
      FP    M 751.0;
      JNB   _00e;
      L     1.000000e+02;
      T     DB70.DBD 52;
_00e: NOP   0;
NETWORK
TITLE =
NETWORK
TITLE =
      A     "OTOMATIK";
      A(;
      L     "JEN2_DATA".STAT11;
      L     1;
      ==I;
      );
      A(;
      L     "AI-SENSOR-DATA".STAT1;
      L     "HMI_DATA".JEN2_Min_Basinc;
      <=R;
      );
      S     "JEN2_DATA".STAT12;
      A     "OTOMATIK";
      A(;
      L     "JEN2_DATA".STAT11;
      L     1;
      ==I;
      );
      A(;
      L     "AI-SENSOR-DATA".STAT1;
      L     "HMI_DATA".JEN2_Max_Basinc;
      >=R;
      );
      R     "JEN2_DATA".STAT12;
      NOP   0;
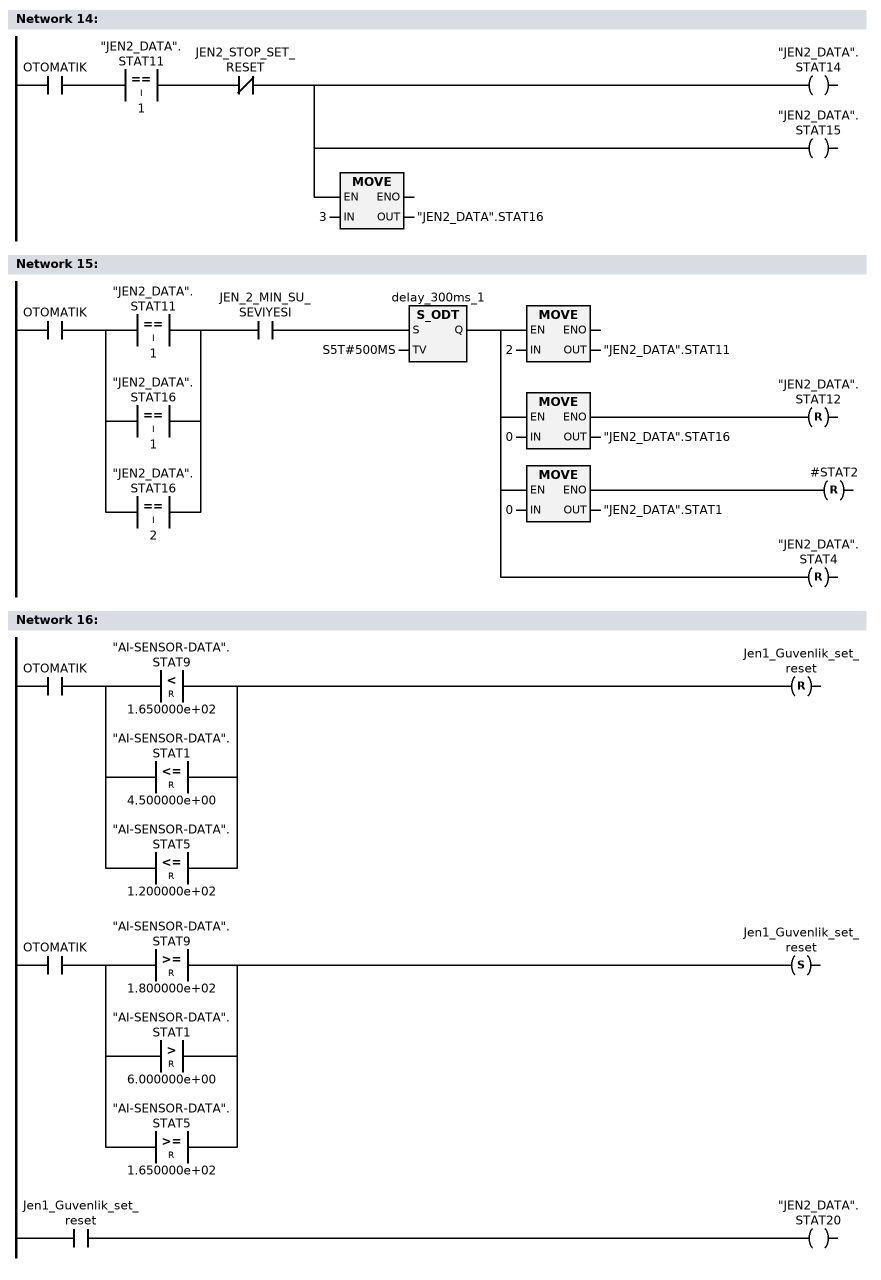
NETWORK
TITLE =
      A     "OTOMATIK";
      A(;
      L     "JEN2_DATA".STAT11;
      L     1;
      ==I;
      );
      AN    "JEN2_STOP_SET_RESET";
      =     L 0.0;
      A     L 0.0;
      BLD   102;
      =     "JEN2_DATA".STAT14;
      A     L 0.0;
      BLD   102;
      =     "JEN2_DATA".STAT15;
      A     L 0.0;
      JNB   _00f;
      L     3;
      T     "JEN2_DATA".STAT16;
_00f: NOP   0;
NETWORK
TITLE =
      A     "OTOMATIK";
      A(;
      O(;
      L     "JEN2_DATA".STAT11;
      L     1;
      ==I;
      );
      O(;
      L     "JEN2_DATA".STAT16;
      L     1;
      ==I;
      );
      O(;
      L     "JEN2_DATA".STAT16;
      L     2;
      ==I;
      );
      );
      A     "JEN_2_MIN_SU_SEVIYESI";
      L     S5T#500MS;
      SD    "delay_300ms_1";
      NOP   0;
      NOP   0;
      NOP   0;
      A     "delay_300ms_1";
      =     L 0.0;
      A     L 0.0;
      JNB   _010;
      L     2;
      T     "JEN2_DATA".STAT11;
_010: NOP   0;
      A     L 0.0;
      JNB   _011;
      L     0;
      T     "JEN2_DATA".STAT16;
      SET;
      SAVE;
      CLR;
_011: A     BR;
      R     "JEN2_DATA".STAT12;
      A     L 0.0;
      JNB   _012;
      L     0;
      T     "JEN2_DATA".STAT1;
      SET;
      SAVE;
      CLR;
_012: A     BR;
      R     #STAT2;
      A     L 0.0;
      BLD   102;
      R     "JEN2_DATA".STAT4;
NETWORK
TITLE =
      A     "OTOMATIK";
      A(;
      O(;
      L     "AI-SENSOR-DATA".STAT9;
      L     1.650000e+02;
      <R;
      );
      O(;
      L     "AI-SENSOR-DATA".STAT1;
      L     4.500000e+00;
      <=R;
      );
      O(;
      L     "AI-SENSOR-DATA".STAT5;
      L     1.200000e+02;
      <=R;
      );
      );
      R     "Jen1_Guvenlik_set_reset";
      A     "OTOMATIK";
      A(;
      O(;
      L     "AI-SENSOR-DATA".STAT9;
      L     1.800000e+02;
      >=R;
      );
      O(;
      L     "AI-SENSOR-DATA".STAT1;
      L     6.000000e+00;
      >R;
      );
      O(;
      L     "AI-SENSOR-DATA".STAT5;
      L     1.650000e+02;
      >=R;
      );
      );
      S     "Jen1_Guvenlik_set_reset";
      A     "Jen1_Guvenlik_set_reset";
      =     "JEN2_DATA".STAT20;
NETWORK
TITLE =
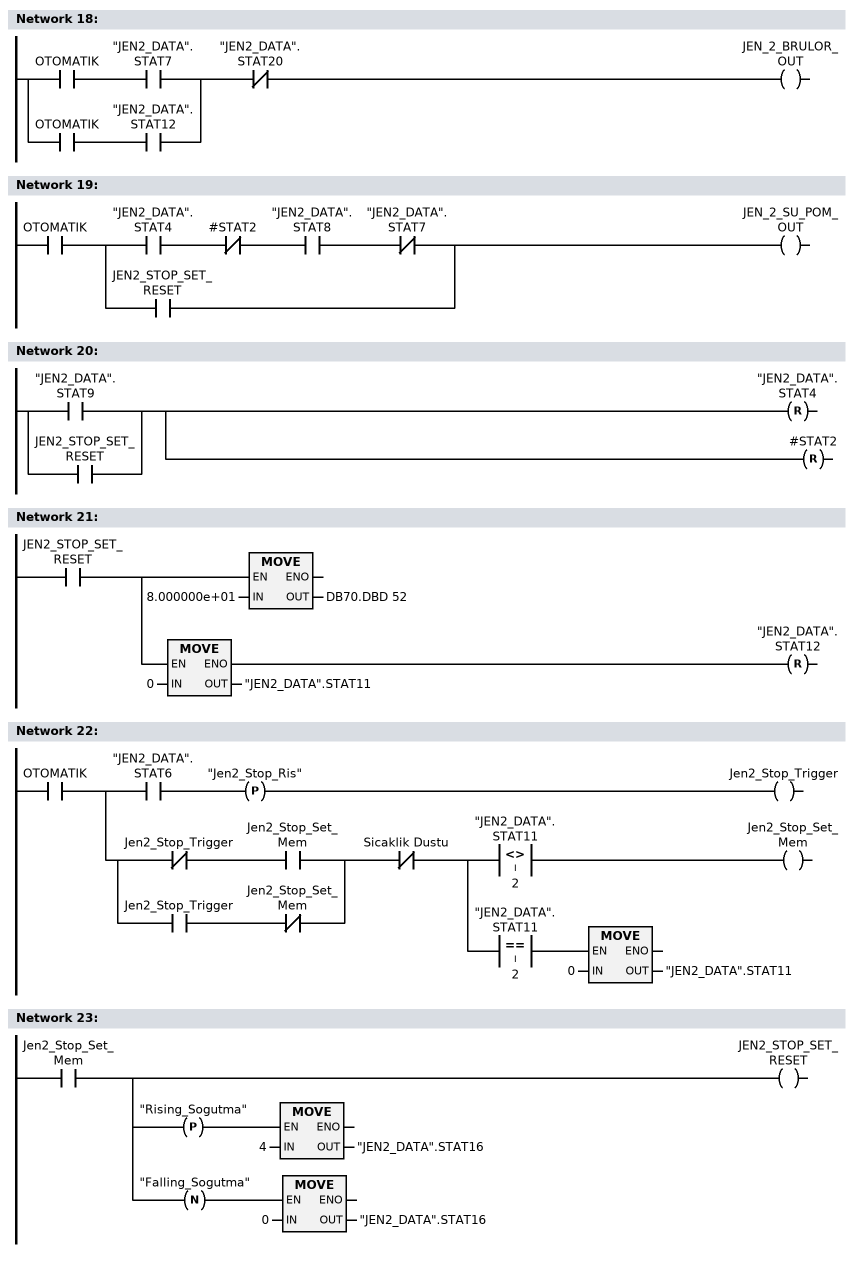
NETWORK
TITLE =
      A(;
      A     "OTOMATIK";
      A     "JEN2_DATA".STAT7;
      O;
      A     "OTOMATIK";
      A     "JEN2_DATA".STAT12;
      );
      AN    "JEN2_DATA".STAT20;
      =     "JEN_2_BRULOR_OUT";
NETWORK
TITLE =
      A     "OTOMATIK";
      A(;
      A     "JEN2_DATA".STAT4;
      AN    #STAT2;
      A     "JEN2_DATA".STAT8;
      AN    "JEN2_DATA".STAT7;
      O     "JEN2_STOP_SET_RESET";
      );
      =     "JEN_2_SU_POM_OUT";
NETWORK
TITLE =
      O     "JEN2_DATA".STAT9;
      O     "JEN2_STOP_SET_RESET";
      R     "JEN2_DATA".STAT4;
      R     #STAT2;
NETWORK
TITLE =
      A     "JEN2_STOP_SET_RESET";
      =     L 0.0;
      A     L 0.0;
      JNB   _013;
      L     8.000000e+01;
      T     DB70.DBD 52;
_013: NOP   0;
      A     L 0.0;
      JNB   _014;
      L     0;
      T     "JEN2_DATA".STAT11;
      SET;
      SAVE;
      CLR;
_014: A     BR;
      R     "JEN2_DATA".STAT12;
NETWORK
TITLE =
      A     "OTOMATIK";
      =     L 0.0;
      A     L 0.0;
      A     "JEN2_DATA".STAT6;
      FP    "Jen2_Stop_Ris";
      =     "Jen2_Stop_Trigger";
      A     L 0.0;
      A(;
      AN    "Jen2_Stop_Trigger";
      A     "Jen2_Stop_Set_Mem";
      O;
      A     "Jen2_Stop_Trigger";
      AN    "Jen2_Stop_Set_Mem";
      );
      AN    "Sicaklik Dustu";
      =     L 0.1;
      A     L 0.1;
      A(;
      L     "JEN2_DATA".STAT11;
      L     2;
      <>I;
      );
      =     "Jen2_Stop_Set_Mem";
      A     L 0.1;
      A(;
      L     "JEN2_DATA".STAT11;
      L     2;
      ==I;
      );
      JNB   _015;
      L     0;
      T     "JEN2_DATA".STAT11;
_015: NOP   0;
NETWORK
TITLE =
      A     "Jen2_Stop_Set_Mem";
      =     L 0.0;
      A     L 0.0;
      BLD   102;
      =     "JEN2_STOP_SET_RESET";
      A     L 0.0;
      FP    "Rising_Sogutma";
      JNB   _016;
      L     4;
      T     "JEN2_DATA".STAT16;
_016: NOP   0;
      A     L 0.0;
      FN    "Falling_Sogutma";
      JNB   _017;
      L     0;
      T     "JEN2_DATA".STAT16;
_017: NOP   0;
